ACTION _mode_manager:
IF process_mode_req_is_pending(prc)
THEN
    process_apply_mode_req_first_step(prc);
    CASE process_get_mode(prc) OF
        MODE_TO_ABSENT:
			;
        MODE_TO_INACTIVE:
			;
        MODE_TO_TEST:
			;
        MODE_TO_OPERATIONAL:
			;
    END_CASE
    process_apply_mode_req_second_step(prc);
END_IF
END_ACTION

ACTION _object_manager:
IF objects_initialization()
THEN
	sub_process_init(
		object_name					:= 'csp_case_closing_os.prc', 
		process						:= csp_case_closing.prc, 
		CONVERSION_this				:= prc);
		
	prc_path 						:= process_get_path(prc);
	
	process_message_init(
        object_name:= CONCAT(prc_path, '_Closing_paddle_Cleanout_position_aem'),
        behaviour:= MESSAGE_BEHAVIOUR_STATE,
        reset_timeout:= 0,
        disableable:= FALSE,
        individual_reset:= FALSE,
        machine_reaction:= MACHINE_REACTION_EMERGENCY_STOP, 
        typology:=  MESSAGE_TYPOLOGY_ABNORMAL,
        process:= prc,
        CONVERSION_this:= Closing_paddle_Cleanout_position_aem);
END_IF

IF objects_running()
THEN
	process_cycle(prc);
END_IF
END_ACTION

ACTION _read_process_image:
;
END_ACTION

ACTION _read_var_input:
;
END_ACTION

ACTION _set_runtime_properties:
;
END_ACTION

ACTION _write_output:
;
END_ACTION

END_PROGRAM

// ---- Application/CSP/Case/Closing/LS/csp_case_closing_ls.TcPOU
(*********************************** G.D S.p.A. - Technical Department ***********************************
============= PROGRAM INFO ============
FOLDER:             TBD
MACHINES INVOLVED:  TBD 

============= DESCRIPTION =============
csp machine declaration

============= REVISIONS ===============
Date		Version	 	Author      	Description             
----------	-------		------------  	--------------------------------------------
2019/04/05 	0000.00	 	M.Grasso		Creation of the PRG

**********************************************************************************************************)
(*$R process_ref := prc; $*)
PROGRAM csp_case_closing_ls
VAR
		
	prc:											process;
	prc_path:										STRING;
	
	phase_upper:									BOOL;
	phase_lower:									BOOL;
	phase_horizontal:								BOOL;
	
	horizontal_first:								BOOL;
	horizontal_second:								BOOL;
	
END_VAR

_read_var_input();

_object_manager();

IF NOT objects_running()
THEN
	RETURN;	
END_IF

_read_process_image();

_mode_manager();

CASE process_get_mode(prc) OF
	MODE_ABSENT,
	MODE_INACTIVE:
		RETURN;
	MODE_TEST:
		_handle_process_test();
END_CASE

_set_runtime_properties();

(********************************* BODY *********************************)

(* CLEARS PHASING SEQUENCE DUE TO AXES CAM ENGAGED *)
IF 	axis_is_cam_engaged(csp_case_closing_ls_horizontal.axis)
	OR machine_is_stop_emergency_active(csp.mch)
THEN
	phase_horizontal := FALSE;
END_IF

IF 	axis_is_cam_engaged(csp_case_closing_ls_upper.axis)
	OR machine_is_stop_emergency_active(csp.mch)
THEN
	phase_upper := FALSE;
END_IF

IF 	axis_is_cam_engaged(csp_case_closing_ls_lower.axis)
	OR machine_is_stop_emergency_active(csp.mch)
THEN
	phase_lower := FALSE;
END_IF

IF (
	axis_is_cam_engaged(csp_case_closing_ls_horizontal.axis)
	AND axis_is_cam_engaged(csp_case_closing_ls_upper.axis)
	AND axis_is_cam_engaged(csp_case_closing_ls_lower.axis)
	)
	OR machine_is_stop_emergency_active(csp.mch)
THEN
	horizontal_first := FALSE;
	horizontal_second := FALSE;
END_IF


(* HORIZONTAL NEEDS TO PHASE - CHECK IF UPPER AND LOWER MOVE FIRST OR HORIZONTAL FIRST *)
IF	NOT axis_is_cam_engaged(csp_case_closing_ls_horizontal.axis)
	AND NOT csp_case_closing_ls_horizontal.phase_done
	AND (motorization_manager_is_starting(csp_main_motorization_manager.motm) OR jog_manager_is_jog_axis_active(JOG_LIST_CSP_CASE_VIRTUAL, csp_main_jogManager.jog_manager_virtual))
THEN	
	(* CALCULATED HORIZONTAL TO MOVE IN - MOVE UPPER AND LOWER FIRST *)
	IF csp_case_closing_ls_horizontal.axis_calculated_cam_slave_position_deg >= axis_get_actual_modulo_position(csp_case_closing_ls_horizontal.axis)
	THEN
		horizontal_second := TRUE;
	(* CALCULATED HORIZONTAL TO MOVE OUT - MOVE HORIZONTAL FIRST *)
	ELSE
		horizontal_first := TRUE;
	END_IF
END_IF

(* PHASE HORIZONTAL THEN UPPER AND LOWER *)
IF 	horizontal_first
	AND (motorization_manager_is_starting(csp_main_motorization_manager.motm) OR jog_manager_is_jog_axis_active(JOG_LIST_CSP_CASE_VIRTUAL, csp_main_jogManager.jog_manager_virtual))
THEN
	phase_horizontal := TRUE;
	IF csp_case_closing_ls_horizontal.phase_done
	THEN
		phase_upper := TRUE;
		phase_lower := TRUE;
	END_IF
END_IF

(* PHASE UPPER AND LOWER THEN HORIZONTAL *)
IF horizontal_second
	AND (motorization_manager_is_starting(csp_main_motorization_manager.motm) OR jog_manager_is_jog_axis_active(JOG_LIST_CSP_CASE_VIRTUAL, csp_main_jogManager.jog_manager_virtual))
THEN
	phase_upper := TRUE;
	phase_lower := TRUE;
	IF 	csp_case_closing_ls_upper.phase_done
		AND csp_case_closing_ls_lower.phase_done
	THEN
		phase_horizontal := TRUE;
	END_IF
END_IF

(************************************************************************)

_handle_messages();

_write_output();

ACTION _handle_messages:
;
END_ACTION

ACTION _handle_process_test:
;
END_ACTION

ACTION _mode_manager:
IF process_mode_req_is_pending(prc)
THEN
    process_apply_mode_req_first_step(prc);
    CASE process_get_mode(prc) OF
        MODE_TO_ABSENT:
			;
        MODE_TO_INACTIVE:
			;
        MODE_TO_TEST:
			;
        MODE_TO_OPERATIONAL:
			;
    END_CASE
    process_apply_mode_req_second_step(prc);
END_IF
END_ACTION

ACTION _object_manager:
IF objects_initialization()
THEN
	sub_process_init(
		object_name					:= 'csp_case_closing_ls.prc', 
		process						:= csp_case_closing.prc, 
		CONVERSION_this				:= prc);
		
	prc_path 						:= process_get_path(prc);
END_IF

IF objects_running()
THEN
	process_cycle(prc);
END_IF
END_ACTION

ACTION _read_process_image:
;
END_ACTION

ACTION _read_var_input:
;
END_ACTION

ACTION _set_runtime_properties:
;
END_ACTION

ACTION _write_output:
;
END_ACTION

END_PROGRAM

// ---- Application/CSP/Case/Discharge/_Tasks/_csp_case_discharge_normal.TcPOU
(*********************************** G.D S.p.A. - Technical Department ***********************************
============= PROGRAM INFO ============
FOLDER:             TBD
MACHINES INVOLVED:  TBD 

============= DESCRIPTION =============
csp main interface program

============= REVISIONS ===============
Date		Version	 	Author      	Description             
----------	-------		------------  	--------------------------------------------
2019/09/27 	0000.00	 	M.Grasso		Creation of the PRG

**********************************************************************************************************)
PROGRAM _csp_case_discharge_normal
VAR
END_VAR

(* CASE *)
	(* DISCHARGE *)
		(* SPEEDBELT *)
		csp_case_discharge_speedBelt();
		(* REJECT *)
		csp_case_discharge_reject();

END_PROGRAM

// ---- Application/CSP/Case/Discharge/Speed Belt/csp_case_discharge_speedBelt.TcPOU
(*********************************** G.D S.p.A. - Technical Department ***********************************
============= PROGRAM INFO ============
FOLDER:             TBD
MACHINES INVOLVED:  TBD 

============= DESCRIPTION =============
csp machine declaration

============= REVISIONS ===============
Date		Version	 	Author      	Description             
----------	-------		------------  	--------------------------------------------
2019/04/05 	0000.00	 	M.Grasso		Creation of the PRG

**********************************************************************************************************)
(*$R process_ref := prc; $*)
PROGRAM csp_case_discharge_speedBelt
VAR
		
	prc:											process;
	prc_path:										STRING;
	
END_VAR

_read_var_input();

_object_manager();

IF NOT objects_running()
THEN
	RETURN;	
END_IF

_read_process_image();

_mode_manager();

_set_runtime_properties();

(********************************* BODY *********************************)
(************************************************************************)

_handle_messages();

_write_output();

ACTION _handle_messages:
;
END_ACTION

ACTION _handle_process_test:
;
END_ACTION

ACTION _mode_manager:
IF process_mode_req_is_pending(prc)
THEN
    process_apply_mode_req_first_step(prc);
    CASE process_get_mode(prc) OF
        MODE_TO_ABSENT:
			;
        MODE_TO_INACTIVE:
			;
        MODE_TO_TEST:
			;
        MODE_TO_OPERATIONAL:
			;
    END_CASE
    process_apply_mode_req_second_step(prc);
END_IF
END_ACTION

ACTION _object_manager:
IF objects_initialization()
THEN
	sub_process_init(
		object_name					:= 'csp_case_discharge_speedBelt.prc', 
		process						:= csp_case_discharge.prc, 
		CONVERSION_this				:= prc);
		
	prc_path 						:= process_get_path(prc);
END_IF

IF objects_running()
THEN
	process_cycle(prc);
END_IF
END_ACTION

ACTION _read_process_image:
;
END_ACTION

ACTION _read_var_input:
;
END_ACTION

ACTION _set_runtime_properties:
;
END_ACTION

ACTION _write_output:
;
END_ACTION

END_PROGRAM

// ---- Application/CSP/Case/Discharge/Reject/csp_case_discharge_reject.TcPOU
(*********************************** G.D S.p.A. - Technical Department ***********************************
============= PROGRAM INFO ============
FOLDER:             TBD
MACHINES INVOLVED:  TBD 

 

============= DESCRIPTION =============
csp machine declaration

 

============= REVISIONS ===============
Date        Version         Author          Description             
----------    -------        ------------      --------------------------------------------
2019/04/05     0000.00         M.Grasso        Creation of the PRG

 

**********************************************************************************************************)
(*$R process_ref := prc; $*)
PROGRAM csp_case_discharge_reject
VAR
        
    prc:                                            	process;
    prc_path:                                        	STRING;
    
    reject_ftrig:                                    	F_TRIG;
    di:                                             	Digital_input;
    reject_active:                                    	BOOL;
    reject_belt_run_delay:                             	Timer;

    status:                                         	STRING;
    start_reject:                                   	BOOL;
	trigger:                                         	BOOL;
	MODSORT_reject:                                 	BOOL;
    MODSORT_fwd:                                     	BOOL;
	reject_confirm:                                 	TON;
	start_reject_belt:                                	BOOL;
    reject_confirmed:                                 	BOOL;
    case_at_reject:                                  	INT:=28;
	open_major_LS_detected: 							BOOL := FALSE;
	open_major_OS_detected:								BOOL := FALSE;

	open_trailing_minor:								BOOL;
	Discharge_reject_count:								DINT;
	timer1:												TOF;
	timer1_value:									TIME := T#5S;
	time_complete1: 									BOOL;
	open_leading_minor: 								BOOL;
	Startup_run_ton: 									Ton;
	startup_run_condition: 								BOOL;
	modsort_belt_speed_analog_reference_ao:             analog_output;
    speed_value_nvr: 									REAL;
	stopping_run_ton: 									Ton;
	stop_run_condition: 								BOOL;
	suspend_run_ton: 									TON;
	suspend_run_condition: 								BOOL;
END_VAR
VAR CONSTANT
    MOTOR_MAX_VELOCITY_DEGPS:                        	LREAL := 9600;
    MOTOR_MIN_VELOCITY_DEGPS:                         	LREAL := 100;
    MOTOR_MAX_ACCELLERATION_DEGPS2:                    	LREAL := 4800;
    MOTOR_MAX_DECELLERATION_DEGPS2:                    	LREAL := 4800;
    MOTOR_MAX_JERK_DEGPS3:                            	LREAL := 100000000; 
    MOTOR_MAX_FOLLOWING_ERROR_DEG:                    	LREAL := 2;
END_VAR

_read_var_input();

 

_object_manager();

 

IF NOT objects_running()
THEN
    RETURN;    
END_IF

 

_read_process_image();

 

_mode_manager();

 

_set_runtime_properties();

 

(********************************* BODY *********************************)
(* Handles stops for reject belt and Modsort Motors to turnoff when machine is not in execute *)
IF  (
	axis_is_moving(csp_main_motorization_virtualManager.axis) 
	OR 
	NOT stop_run_condition
	)
	AND NOT csp.o_machine_is_emergency_stopped
THEN 
 	speed_value_nvr := csp_main_motorization_manager.motm.actual_velocity * 200;
ELSE
	speed_value_nvr := 0;
END_IF

analog_output_electrical_write(
    electrical_value := speed_value_nvr,
    conversion_THIS := modsort_belt_speed_analog_reference_ao);
 
IF 	reject_confirmed
THEN
    modsort_reject := FALSE;
    digital_output_reset(conversion_this:= csp_case_discharge_reject_modsort.MODSORT_REJECT_RUN_do); //stops modosort when machine is stopped
END_IF

(*Latches in open flap detected when in window and open flap PE is blocked *)
IF 	((csp_case_virtualMaster.axis.actual_position > csp_case_openFlap_sensors.OpenMajorFlapChkBeginPhase)
	AND
	(csp_case_virtualMaster.axis.actual_position < csp_case_openFlap_sensors.OpenMajorFlapChkEndPhase))
THEN
	IF	NOT digital_input_is_active(csp_case_openFlap_sensors.open_flap_ls_di)
	THEN
		open_major_LS_detected :=TRUE;
	END_IF
	
	IF	NOT digital_input_is_active(csp_case_openFlap_sensors.open_flap_os_di)
	THEN
		open_major_OS_detected :=TRUE;
	END_IF
 END_IF
 
 
(* Resets open flap detected latch *)
IF 	open_major_LS_detected
 	AND axis_get_actual_modulo_position(csp_case_transport_virtualMaster.axis) > 350 //resets open major detected before next case
THEN
	open_major_LS_detected := FALSE;
END_IF

(* Resets open flap detected latch *)
IF 	open_major_OS_detected
 	AND axis_get_actual_modulo_position(csp_case_transport_virtualMaster.axis) > 350 //resets open major detected before next case
THEN
	open_major_OS_detected := FALSE;
END_IF

(* LATCHES BIT FOR OPEN TRAILING MINOR *)
IF 	csp_case_transport_virtualMaster.axis.actual_position > csp_case_openFlap_sensors.open_trailing_minor_begin_phase
	AND csp_case_transport_virtualMaster.axis.actual_position < csp_case_openFlap_sensors.open_trailing_minor_end_phase
THEN
	IF digital_input_is_active(csp_case_openFlap_sensors.open_trailing_minor_di)
	THEN
		open_trailing_minor := TRUE;
	END_IF
END_IF

(* Resets open trailing minor detected latch *)
IF 	open_trailing_minor
	AND axis_get_actual_modulo_position(csp_case_transport_virtualMaster.axis) > 350 //resets open major detected before next case
THEN
 	open_trailing_minor := FALSE;
END_IF

(* LATCHES BIT FOR OPEN LEADING MINOR *)
IF 	csp_case_transport_virtualMaster.axis.actual_position > csp_case_openFlap_sensors.open_leading_minor_begin_phase
	AND csp_case_transport_virtualMaster.axis.actual_position < csp_case_openFlap_sensors.open_leading_minor_end_phase
THEN
	IF digital_input_is_active(csp_case_openFlap_sensors.open_trailing_minor_di)
	THEN
		open_leading_minor := TRUE;
	END_IF
END_IF

(* Resets open OPEN LEADING MINOR detected latch *)
IF 	open_leading_minor
	AND axis_get_actual_modulo_position(csp_case_transport_virtualMaster.axis) > 350 //resets open major detected before next case
THEN
 	open_leading_minor := FALSE;
END_IF

(* Sets shift register if detected *)
IF open_trailing_minor
THEN
	shift_register_step_set_reject_reason(
		reject_reason_to_set := TRAILING_MINOR_FLAP_OPEN,
		step_id := 28,
		CONVERSION_this := csp_case_main_statistics.sr);
END_IF

(* Sets shift register if detected *)
IF 	open_leading_minor
THEN
	shift_register_step_set_reject_reason(
		reject_reason_to_set := LEADING_MINOR_FLAP_OPEN,
		step_id := 28,
		CONVERSION_this := csp_case_main_statistics.sr);
END_IF

(* Sets shift register if detected *)
IF 	open_major_LS_detected
THEN
	shift_register_step_set_reject_reason(
		reject_reason_to_set := OPEN_FLAP_LOADER_SIDE,
		step_id := 28,
		CONVERSION_this := csp_case_main_statistics.sr);
END_IF

(* Sets shift register if detected *)
IF 	open_major_OS_detected
THEN	
	shift_register_step_set_reject_reason(
		reject_reason_to_set := OPEN_FLAP_OPERATOR_SIDE,
		step_id := 28,
		CONVERSION_this := csp_case_main_statistics.sr);
END_IF

(* Shift Register detects if there is a reject *)
IF shift_register_step_has_any_reject_reason(
	step_id:= case_at_reject, 
	CONVERSION_this:= csp_case_main_statistics.sr)
THEN
	reject_active := TRUE;
ELSE
	reject_active:= FALSE;
END_IF
             
digital_input_read(trigger, csp_case_discharge_reject_sensors.reject_trigger_di); // sets 'trigger' as bool for digital input OF PhotoEye

reject_ftrig(CLK := trigger); // falling edge of trigger //starts reject on trigger if reject_active (ON)

reject_confirm(IN:=start_reject , PT:=T#2S , Q=> reject_confirmed , ET=> );// how long to run reject operation or setup with Photoeye for confirmation

IF reject_active AND reject_ftrig.Q    //start sequence when PE triggered
THEN
	start_reject := TRUE;
END_IF
    
(* Resets start_reject to end the reject sequence *)    
IF reject_confirmed 
THEN     (*resets bit when reject confirmed (2 Second Timer); works for max speed at 27.5 cpm with cycle being 2.18 seconds *)
    start_reject := FALSE;    
END_IF            

(********************************* MODSORT LOGIC *********************************)
stopping_run_ton(IN:= NOT axis_is_moving(csp_main_motorization_virtualManager.axis) , PT:=T#10S , Q=> stop_run_condition , ET=> );
suspend_run_ton(
				IN:= motorization_manager_is_held(csp_main_motorization_manager.motm) OR motorization_manager_is_suspended(csp_main_motorization_manager.motm),
				PT:=T#20S,
				Q=> suspend_run_condition,
				ET=> );
 
IF 	(
		(
			axis_is_moving(csp_main_motorization_virtualManager.axis) 
			OR
			NOT stop_run_condition //becomes true after moto VM stopped for 2 seconds
		)
		AND NOT suspend_run_condition //becomes true after 5 seconds of being in suspend or held state
	)
	AND NOT csp.o_machine_is_emergency_stopped
THEN
	IF digital_output_is_active(conversion_this:= csp_case_discharge_reject_modsort.MODSORT_REJECT_RUN_do)
	THEN
		digital_output_reset(conversion_this:= csp_case_discharge_reject_modsort.MODSORT_FWD_RUN_do);
		modsort_fwd := FALSE; //testing
	ELSE
		modsort_fwd := TRUE; //testing
		digital_output_set(conversion_this:= csp_case_discharge_reject_modsort.MODSORT_FWD_RUN_do);
	END_IF    
ELSE
	modsort_fwd := FALSE; //testing
	digital_output_reset(conversion_this:= csp_case_discharge_reject_modsort.MODSORT_FWD_RUN_do);
END_IF

(* If reject sequence activated, and machine running, then run modsort reject motor until confirmed with (2 second) timer.*)    
IF 	reject_active 
	AND start_reject 
	AND NOT reject_confirmed    //reject once started until reject_confirm TRUE
THEN
	modsort_reject := TRUE;
	digital_output_set(conversion_this:= csp_case_discharge_reject_modsort.MODSORT_REJECT_RUN_do);
END_IF    
    
start_reject_belt := reject_active//start_reject                             //conditions for starting reject belt
                    OR digital_output_is_active(conversion_this:= csp_case_discharge_reject_modsort.MODSORT_REJECT_RUN_do);          
        

(********************************* Belt Run duration *********************************)
							
timer1.IN := trigger;
time_complete1 := NOT timer1.Q;
timer1(PT := timer1_value);

(********************************* REJECT BELT LOGIC *********************************)
Startup_run_ton(IN:=axis_is_moving(csp_main_motorization_virtualManager.axis) , PT:=T#5S , Q=> startup_run_condition , ET=> );

IF 	(
		start_reject_belt 
		AND NOT time_complete1
	)
	OR
	(
		axis_is_moving(csp_main_motorization_virtualManager.axis)
		AND NOT startup_run_condition
	)
THEN
	axis_set_override(                        //overides axis velocity to the set JOG speed, JOG set at 10 in csp_case_discharge_belts_conveyor (TEST SPEED - Austin)
		speed_override_percent     := 30,
		CONVERSION_this         := csp_case_discharge_reject_belt.axis);//csp_case_discharge_belts_conveyor.axis
	status := 'Belt moving';
ELSE
	axis_set_override(          
		speed_override_percent     := 0,
		CONVERSION_this         := csp_case_discharge_reject_belt.axis);
	status := 'Stopped';
END_IF


(************************************************************************)

Discharge_Reject_Count :=
(
csp_case_main_statistics.logsect.hmi_shift_independent_sampled_counters.reject_reasons_counters[16]
+
csp_case_main_statistics.logsect.hmi_shift_independent_sampled_counters.reject_reasons_counters[17]
+
csp_case_main_statistics.logsect.hmi_shift_independent_sampled_counters.reject_reasons_counters[18]
+
csp_case_main_statistics.logsect.hmi_shift_independent_sampled_counters.reject_reasons_counters[19]
+
csp_case_main_statistics.logsect.hmi_shift_independent_sampled_counters.reject_reasons_counters[20]
+
csp_case_main_statistics.logsect.hmi_shift_independent_sampled_counters.reject_reasons_counters[21]
+
csp_case_main_statistics.logsect.hmi_shift_independent_sampled_counters.reject_reasons_counters[22]
+
csp_case_main_statistics.logsect.hmi_shift_independent_sampled_counters.reject_reasons_counters[23]
+
csp_case_main_statistics.logsect.hmi_shift_independent_sampled_counters.reject_reasons_counters[24]
);
(************************************************************************)


 

_handle_messages();

 

_write_output();

ACTION _handle_messages:
;
END_ACTION

ACTION _handle_process_test:
;
END_ACTION

ACTION _mode_manager:
IF process_mode_req_is_pending(prc)
THEN
    process_apply_mode_req_first_step(prc);
    CASE process_get_mode(prc) OF
        MODE_TO_ABSENT:
			;
        MODE_TO_INACTIVE:
			;
        MODE_TO_TEST:
			;
        MODE_TO_OPERATIONAL:
			;
    END_CASE
    process_apply_mode_req_second_step(prc);
END_IF
END_ACTION

ACTION _object_manager:
IF objects_initialization()
THEN
	sub_process_init(
		object_name					:= 'csp_case_discharge_reject.prc', 
		process						:= csp_case_discharge.prc, 
		CONVERSION_this				:= prc);
		
	prc_path 						:= process_get_path(prc);
	
	timer_init(
    	object_name:= 'csp_case_discharge_reject.reject_belt_run_delay',
    	process:= prc,
    	conversion_THIS:= reject_belt_run_delay);

 analog_output_init(
            object_name            	:= '_modsort_belt_speed_analog_reference_ao',
            field_min            	:= 0,                                (* Campo lettura modulo Beckhoff, unità - min value *)
            field_max             	:= MAX_INT_VALUE,                    (* Campo lettura modulo Beckhoff, unità - max value *)
            field_ele_xa        	:= 0,
            field_ele_ya        	:= 0,
            field_ele_xb        	:= MAX_INT_VALUE,
            field_ele_yb        	:= 10000,
            electrical_min        	:= 0,                                (* Saturazione - valore minimo in uscita, mV *)
            electrical_max        	:= 10000,                            (* Saturazione - valore massimo in uscita, mV *)
            ele_phy_xa           	:= 0,        (* mV *)
            ele_phy_ya            	:= 0,        (* PPM *)
            ele_phy_xb            	:= 10000,    (* mV *)
            ele_phy_yb            	:= 10000,    (* PPM *)
            physical_min        	:= 0,        (* rpm *)
            physical_max         	:= 5000,    (* rpm *)
            process                	:= prc,
            conversion_THIS         := modsort_belt_speed_analog_reference_ao
            ); 
END_IF

IF objects_running()
THEN
	process_cycle(prc);
    analog_output_cycle(conversion_THIS := modsort_belt_speed_analog_reference_ao);
END_IF
END_ACTION

ACTION _read_process_image:
;
END_ACTION

ACTION _read_var_input:
;
END_ACTION

ACTION _set_runtime_properties:
;
END_ACTION

ACTION _write_output:
;
END_ACTION

END_PROGRAM

// ---- Application/CSP/Case/Open Flap/Sensors/csp_case_openFlap_sensors.TcPOU
(*********************************** G.D S.p.A. - Technical Department ***********************************
============= PROGRAM INFO ============
FOLDER:             TBD
MACHINES INVOLVED:  TBD 

============= DESCRIPTION =============
csp machine declaration

============= REVISIONS ===============
Date		Version	 	Author      	Description             
----------	-------		------------  	--------------------------------------------
2019/04/05 	0000.00	 	M.Grasso		Creation of the PRG

**********************************************************************************************************)
(*$R process_ref := prc; $*)
PROGRAM csp_case_openFlap_sensors
VAR
	
	prc:											process;
	prc_path:										STRING;
	
	open_flap_ls_di:								digital_input;
	open_flap_os_di:								digital_input;
		
	open_major_flap_os_di_dchk: 					check_section;
	open_major_flap_ls_di_dchk: 					check_section;
	
	
	open_trailing_minor_di:							digital_input;
	open_trailing_minor_chksect:					check_section;
	open_trailing_minor_begin_phase: 				LREAL := 170; (*$P $*)
	open_trailing_minor_end_phase:					LREAL := 188; (*$P $*)
	
	open_leading_minor_chksect:						check_section;
	open_leading_minor_begin_phase: 				LREAL := 90; (*$P $*)
	open_leading_minor_end_phase:					LREAL := 110; (*$P $*)
	
	quality_reject_dchk: 							check_section;
	quality_reject_bool: 							boolean;
	quality_reject_req:								BOOL:= FALSE; (*$P $*)
	quality_reject_aem:								message;
	
	incomplete_glue_reject_dchk: 					check_section;
	incomplete_glue_reject_bool: 					boolean;
	incomplete_glue_reject_aem:						message;
	incomplete_glue_begin_phase: 					LREAL := 10; (*$P $*)
	incomplete_glue_end_phase:						LREAL := 300; (*$P $*)
	
	
	OpenMajorFlapChkBeginPhase: 					LREAL :=100;(*$P $*)
	OpenMajorFlapChkEndPhase:						LREAL :=350;(*$P $*)
	majorFlap_os_inchoerence_chksect: 				check_section;
	majorFlap_ls_inchoerence_chksect: 				check_section;
	
	incomplete_glue_reject: 						BOOL;
	check_step_nvr: 								DINT := 26;
	
	detect_next_case_edges: 						BOOL;(*$P desc:= DETECT LEADING AND TRAILING PHASE OF NEXT CASE; $*)
	eye_test_temp: 									BOOL;
	detected_case_leading_edge: 					LREAL;(*$P desc:= DETECTED LEADING PHASE OF CASE; $*)
	detected_case_trailing_edge: 					LREAL;(*$P desc:= DETECTED TRAILING PHASE OF CASE; $*)
END_VAR

_read_var_input();

_object_manager();

IF NOT objects_running()
THEN
	RETURN;	
END_IF

_read_process_image();

_mode_manager();

_set_runtime_properties();

(********************************* BODY *********************************)
check_section_set_check_window_phases_value(
    begin_phase         :=  OpenMajorFlapChkBeginPhase,
    end_phase           :=  OpenMajorFlapChkEndPhase,
    conversion_THIS     :=  open_major_flap_os_di_dchk);

check_section_set_check_window_phases_value(
    begin_phase         :=  OpenMajorFlapChkBeginPhase,
    end_phase           :=  OpenMajorFlapChkEndPhase,
    conversion_THIS     :=  open_major_flap_ls_di_dchk);	
	
	
check_section_set_check_window_phases_value(
    begin_phase         :=  open_trailing_minor_begin_phase,
    end_phase           :=  open_trailing_minor_end_phase,
    conversion_THIS     :=  open_trailing_minor_chksect);	

check_section_set_check_window_phases_value(
    begin_phase         :=  open_leading_minor_begin_phase,
    end_phase           :=  open_leading_minor_end_phase,
    conversion_THIS     :=  open_leading_minor_chksect);		
	
IF quality_reject_req //quality check pb on hmi to reject a case for inspection. Uses checksection to look for pb and then trigger the reject
THEN
	boolean_set(quality_reject_bool);
ELSE
	boolean_reset(quality_reject_bool);
END_IF

//checks for motion and Emergency stop to reject 
check_section_set_check_window_phases_value(
	begin_phase := incomplete_glue_begin_phase,
	end_phase := incomplete_glue_end_phase,
	CONVERSION_this := incomplete_glue_reject_dchk); 

IF check_section_get_step(incomplete_glue_reject_dchk) <> check_step_nvr
THEN
	check_section_set_step(check_step_nvr, incomplete_glue_reject_dchk);
END_IF

IF 	axis_get_actual_modulo_position(csp_case_transport_virtualMaster.axis) > incomplete_glue_begin_phase  
	AND axis_get_actual_modulo_position(csp_case_transport_virtualMaster.axis) < incomplete_glue_end_phase  
	AND machine_is_stop_emergency_active(csp.mch)
THEN
	boolean_set(incomplete_glue_reject_bool);
	incomplete_glue_reject := TRUE ;
END_IF

IF axis_get_actual_modulo_position(csp_case_transport_virtualMaster.axis) > 359
THEN
	boolean_reset(incomplete_glue_reject_bool);
	incomplete_glue_reject := FALSE ;
END_IF

IF csp_case_main_services.dry_cycle_mode
	OR csp_main_motorization.empty_command
THEN
	check_section_disable(majorFlap_os_inchoerence_chksect);
	check_section_disable(majorFlap_ls_inchoerence_chksect);
	check_section_disable(open_major_flap_os_di_dchk);
	check_section_disable(open_major_flap_ls_di_dchk);
	check_section_disable(open_trailing_minor_chksect);
	check_section_disable(open_leading_minor_chksect);
ELSE
	check_section_enable(majorFlap_os_inchoerence_chksect);
	check_section_enable(majorFlap_ls_inchoerence_chksect);
	check_section_enable(open_major_flap_os_di_dchk);
	check_section_enable(open_major_flap_ls_di_dchk);
	check_section_enable(open_trailing_minor_chksect);
	check_section_enable(open_leading_minor_chksect);
END_IF		


IF quality_reject_req
THEN
	process_message_set(1, 1, 1, quality_reject_aem);
ELSE
	process_message_reset(quality_reject_aem);
END_IF

(* Turn on eye_test to capture the leading and trailing edge of the box as it passes open-flap eye. Use these values to then set appropriate phase window values for open flap detection. *)
IF 	detect_next_case_edges
	AND NOT eye_test_temp
	AND digital_input_is_active(open_trailing_minor_di)
then
	detected_case_leading_edge := csp_case_transport_virtualMaster.axis.actual_position;
	eye_test_temp := TRUE;
	detect_next_case_edges := FALSE;
end_if

IF 	eye_test_temp
	AND NOT digital_input_is_active(open_trailing_minor_di)
then
	detected_case_trailing_edge := csp_case_transport_virtualMaster.axis.actual_position;
	eye_test_temp := FALSE;
end_if
(************************************************************************)

_handle_messages();

_write_output();

ACTION _handle_messages:
;
END_ACTION

ACTION _handle_process_test:
;
END_ACTION

ACTION _mode_manager:
IF process_mode_req_is_pending(prc)
THEN
    process_apply_mode_req_first_step(prc);
    CASE process_get_mode(prc) OF
        MODE_TO_ABSENT:
			;
        MODE_TO_INACTIVE:
			;
        MODE_TO_TEST:
			;
        MODE_TO_OPERATIONAL:
			;
    END_CASE
    process_apply_mode_req_second_step(prc);
END_IF
END_ACTION

ACTION _object_manager:
IF objects_initialization()
THEN
    sub_process_init(
        object_name                    := 'csp_case_openFlap_sensors.prc',
        process                        := csp_case_openFlap.prc,
        CONVERSION_this                := prc);
       
    prc_path                         := process_get_path(prc);
   
    (* INPUTS *)
    digital_input_init(
        object_name                    := CONCAT(prc_path, '_open_flap_ls_di'),
        polarity_direct                := TRUE,
        process                        := prc,
        CONVERSION_this                := open_flap_ls_di);
       
    digital_input_init(
        object_name                    := CONCAT(prc_path, '_open_flap_os_di'),
        polarity_direct                := TRUE,
        process                        := prc,
        CONVERSION_this                := open_flap_os_di);
		
	digital_input_init(
        object_name                    := CONCAT(prc_path, '_open_trailing_minor_di'),
        polarity_direct                := TRUE,
        process                        := prc,
        CONVERSION_this                := open_trailing_minor_di);
  
		
	 boolean_init(
		object_name 				   := CONCAT(prc_path, '_quality_reject_bool'),
		process 			   		   := prc,
		CONVERSION_this				   := quality_reject_bool);
	
	 boolean_init(
		object_name 				   := CONCAT(prc_path, '_incomplete_glue_reject_bool'),
		process 					   := prc,
		CONVERSION_this				   := incomplete_glue_reject_bool);

		
		
(*OPEN FLAP OPERATOR SIDE SENSOR LOGIC*)  
	check_section_window_mode_init(
		object_name:= CONCAT(prc_path, '_open_major_flap_os_di_dchk'),
		check_enable:= TRUE, 
		event_to_check:= CHECK_SECTION_EVENT_INPUT_OFF, 
		execution_mode:= CHECK_SECTION_EXECUTION_WHEN_EVENT_OCCURRED, 
		diagnostic_enable:= FALSE, 
		status_bits_to_be_true:= ITEM_CASE_FEED, 
		status_bits_to_be_false:= 0, 
		_step_status_conditioning_execution:= FALSE, 
		status_bits_to_set:= OPEN_FLAP_OPERATOR_SIDE, 
		status_bits_to_reset:= 0, 
		reject_bit_to_set:= OPEN_FLAP_OPERATOR_SIDE, 
		_step:= 28, 
		first_step_to_write_offset:= 0, 
		number_of_steps_to_write:= 1, 
		begin_phase:= OpenMajorFlapChkBeginPhase, 
		end_phase:= OpenMajorFlapChkEndPhase, 
		max_consecutive_failed_checks:= 3, 
		max_failed_checks_percentage:= 100, 
		products_for_failed_checks_percentage:= 10, 
		shift_register:= csp_case_main_statistics.sr , 
		process:= prc, 
		CONVERSION_this:= open_major_flap_os_di_dchk );

	check_section_add_di_input(
		di_input := open_flap_os_di,
		CONVERSION_this:= open_major_flap_os_di_dchk);
	
	message_configure(
        individual_reset                    := FALSE,
        machine_reaction                    := MACHINE_REACTION_STOP_IN_PHASE_ONE,
        typology                            := MESSAGE_TYPOLOGY_ABNORMAL,
        CONVERSION_this                     := open_major_flap_os_di_dchk.too_many_failed_checks_aem.message );	
	
	
 (*OPEN FLAP LOADER SIDE SENSOR LOGIC*)  
	check_section_window_mode_init(
		object_name:= CONCAT(prc_path, '_open_major_flap_ls_di_dchk'),
		check_enable:= TRUE, 
		event_to_check:= CHECK_SECTION_EVENT_INPUT_OFF, 
		execution_mode:= CHECK_SECTION_EXECUTION_WHEN_EVENT_OCCURRED, 
		diagnostic_enable:= FALSE, 
		status_bits_to_be_true:= ITEM_CASE_FEED, 
		status_bits_to_be_false:= 0, 
		_step_status_conditioning_execution:= FALSE, 
		status_bits_to_set:= OPEN_FLAP_LOADER_SIDE, 
		status_bits_to_reset:= 0, 
		reject_bit_to_set:= OPEN_FLAP_LOADER_SIDE, 
		_step:= 28, 
		first_step_to_write_offset:= 0, 
		number_of_steps_to_write:= 1, 
		begin_phase:= OpenMajorFlapChkBeginPhase, 
		end_phase:= OpenMajorFlapChkEndPhase, 
		max_consecutive_failed_checks:= 3, 
		max_failed_checks_percentage:= 100, 
		products_for_failed_checks_percentage:= 10, 
		shift_register:= csp_case_main_statistics.sr , 
		process:= prc, 
		CONVERSION_this:= open_major_flap_ls_di_dchk );

	check_section_add_di_input(
		di_input := open_flap_ls_di,
		CONVERSION_this:= open_major_flap_ls_di_dchk);	
    
	message_configure(
        individual_reset                    := FALSE,
        machine_reaction                    := MACHINE_REACTION_STOP_IN_PHASE_ONE,
        typology                            := MESSAGE_TYPOLOGY_ABNORMAL,
        CONVERSION_this                     := open_major_flap_ls_di_dchk.too_many_failed_checks_aem.message );	
	
    
	(*Quality Reject SENSOR LOGIC*)  //added for quality reject push button on hmi
	check_section_window_mode_init(
		object_name:= CONCAT(prc_path, '_quality_reject_dchk'),
		check_enable:= TRUE, 
		event_to_check:= CHECK_SECTION_EVENT_INPUT_ON, 
		execution_mode:= CHECK_SECTION_EXECUTION_WHEN_EVENT_OCCURRED, 
		diagnostic_enable:= FALSE, 
		status_bits_to_be_true:= ITEM_CASE_FEED, 
		status_bits_to_be_false:= 0, 
		_step_status_conditioning_execution:= FALSE, 
		status_bits_to_set:= 0, 
		status_bits_to_reset:= 0, 
		reject_bit_to_set:= QUALITY_REJECT, 
		_step:= 28, 
		first_step_to_write_offset:= 0, 
		number_of_steps_to_write:= 1, 
		begin_phase:= 10, 
		end_phase:= 340, 
		max_consecutive_failed_checks:= 3, 
		max_failed_checks_percentage:= 100, 
		products_for_failed_checks_percentage:= 10, 
		shift_register:= csp_case_main_statistics.sr , 
		process:= prc, 
		CONVERSION_this:= quality_reject_dchk );

	check_section_add_boolean_input(
		boolean_input:= quality_reject_bool,
		CONVERSION_this:= quality_reject_dchk);	
		
	message_configure(
        individual_reset                    := FALSE,
        machine_reaction                    := MACHINE_REACTION_STOP_IN_PHASE_ONE,
        typology                            := MESSAGE_TYPOLOGY_ABNORMAL,
        CONVERSION_this                     := quality_reject_dchk.too_many_failed_checks_aem.message );		
		
	
check_section_window_mode_init(
		object_name:= CONCAT(prc_path, '_majorFlap_os_inchoerence_chksect'),
		check_enable:= TRUE, 
		event_to_check:= CHECK_SECTION_EVENT_INPUT_ALWAYS_ON, 
		execution_mode:= CHECK_SECTION_EXECUTION_WHEN_EVENT_NOT_OCCURRED, 
		diagnostic_enable:= FALSE, 
		status_bits_to_be_true:= ITEM_CASE_FEED, 
		status_bits_to_be_false:= 0, 
		_step_status_conditioning_execution:= FALSE, 
		status_bits_to_set:= 0, 
		status_bits_to_reset:= 0, 
		reject_bit_to_set:= OPEN_FLAP_OPERATOR_SIDE_INCHOERENCE, 
		_step:= 28, 
		first_step_to_write_offset:= 0, 
		number_of_steps_to_write:= 1, 
		begin_phase:= csp_case_flapControl.Flap_check_begin_phase, 
		end_phase:= csp_case_flapControl.Flap_check_end_phase, 
		max_consecutive_failed_checks:= 3, 
		max_failed_checks_percentage:= 100, 
		products_for_failed_checks_percentage:= 99, 
		shift_register:= csp_case_main_statistics.sr , 
		process:= prc, 
		CONVERSION_this:= majorFlap_os_inchoerence_chksect );

	check_section_add_di_input(
		di_input := open_flap_os_di,
		CONVERSION_this:= majorFlap_os_inchoerence_chksect);

	message_configure(
        individual_reset                    := FALSE,
        machine_reaction                    := MACHINE_REACTION_STOP_IN_PHASE_ONE,
        typology                            := MESSAGE_TYPOLOGY_ABNORMAL,
        CONVERSION_this                     := majorFlap_os_inchoerence_chksect.too_many_failed_checks_aem.message );	
		
    check_section_window_mode_init(
		object_name:= CONCAT(prc_path, '_majorFlap_ls_inchoerence_chksect'),
		check_enable:= TRUE, 
		event_to_check:= CHECK_SECTION_EVENT_INPUT_ALWAYS_ON, 
		execution_mode:= CHECK_SECTION_EXECUTION_WHEN_EVENT_NOT_OCCURRED, 
		diagnostic_enable:= FALSE, 
		status_bits_to_be_true:= ITEM_CASE_FEED, 
		status_bits_to_be_false:= 0, 
		_step_status_conditioning_execution:= FALSE, 
		status_bits_to_set:= 0, 
		status_bits_to_reset:= 0, 
		reject_bit_to_set:= OPEN_FLAP_LOADER_SIDE_INCHOERENCE, 
		_step:= 28, 
		first_step_to_write_offset:= 0, 
		number_of_steps_to_write:= 1, 
		begin_phase:= csp_case_flapControl.Flap_check_begin_phase, 
		end_phase:= csp_case_flapControl.Flap_check_end_phase, 
		max_consecutive_failed_checks:= 3, 
		max_failed_checks_percentage:= 100, 
		products_for_failed_checks_percentage:= 99, 
		shift_register:= csp_case_main_statistics.sr , 
		process:= prc, 
		CONVERSION_this:= majorFlap_ls_inchoerence_chksect );

	check_section_add_di_input(
		di_input := open_flap_ls_di,
		CONVERSION_this:= majorFlap_ls_inchoerence_chksect);
		
	message_configure(
        individual_reset                    := FALSE,
        machine_reaction                    := MACHINE_REACTION_STOP_IN_PHASE_ONE,
        typology                            := MESSAGE_TYPOLOGY_ABNORMAL,
        CONVERSION_this                     := majorFlap_ls_inchoerence_chksect.too_many_failed_checks_aem.message );		
		
	
	(* OPEN TRAILING MINOR LOGIC *)
	check_section_window_mode_init(
		object_name:= CONCAT(prc_path, '_open_trailing_minor_chksect'),
		check_enable:= TRUE, 
		event_to_check:= CHECK_SECTION_EVENT_INPUT_ALWAYS_OFF, 
		execution_mode:= CHECK_SECTION_EXECUTION_WHEN_EVENT_NOT_OCCURRED, 
		diagnostic_enable:= FALSE, 
		status_bits_to_be_true:= ITEM_CASE_FEED, 
		status_bits_to_be_false:= 0, 
		_step_status_conditioning_execution:= FALSE, 
		status_bits_to_set:= 0, 
		status_bits_to_reset:= 0, 
		reject_bit_to_set:= TRAILING_MINOR_FLAP_OPEN, 
		_step:= 28, 
		first_step_to_write_offset:= 0, 
		number_of_steps_to_write:= 1, 
		begin_phase:= open_trailing_minor_begin_phase, 
		end_phase:= open_trailing_minor_end_phase, 
		max_consecutive_failed_checks:= 3, 
		max_failed_checks_percentage:= 100, 
		products_for_failed_checks_percentage:= 99, 
		shift_register:= csp_case_main_statistics.sr , 
		process:= prc, 
		CONVERSION_this:= open_trailing_minor_chksect);

	check_section_add_di_input(
		di_input := open_trailing_minor_di,
		CONVERSION_this:= open_trailing_minor_chksect);
	
	message_configure(
        individual_reset                    := FALSE,
        machine_reaction                    := MACHINE_REACTION_STOP_IN_PHASE_ONE,
        typology                            := MESSAGE_TYPOLOGY_ABNORMAL,
        CONVERSION_this                     := open_trailing_minor_chksect.too_many_failed_checks_aem.message );	
	
	(* OPEN LEADING MINOR LOGIC *)
	check_section_window_mode_init(
		object_name:= CONCAT(prc_path, '_open_leading_minor_chksect'),
		check_enable:= TRUE, 
		event_to_check:= CHECK_SECTION_EVENT_INPUT_ALWAYS_OFF, 
		execution_mode:= CHECK_SECTION_EXECUTION_WHEN_EVENT_NOT_OCCURRED, 
		diagnostic_enable:= FALSE, 
		status_bits_to_be_true:= ITEM_CASE_FEED, 
		status_bits_to_be_false:= 0, 
		_step_status_conditioning_execution:= FALSE, 
		status_bits_to_set:= 0, 
		status_bits_to_reset:= 0, 
		reject_bit_to_set:= LEADING_MINOR_FLAP_OPEN, 
		_step:= 28, 
		first_step_to_write_offset:= 0, 
		number_of_steps_to_write:= 1, 
		begin_phase:= open_leading_minor_begin_phase, 
		end_phase:= open_leading_minor_end_phase, 
		max_consecutive_failed_checks:= 3, 
		max_failed_checks_percentage:= 100, 
		products_for_failed_checks_percentage:= 99, 
		shift_register:= csp_case_main_statistics.sr , 
		process:= prc, 
		CONVERSION_this:= open_leading_minor_chksect);

	check_section_add_di_input(
		di_input := open_trailing_minor_di,
		CONVERSION_this:= open_leading_minor_chksect); 
    
	message_configure(
        individual_reset                    := FALSE,
        machine_reaction                    := MACHINE_REACTION_STOP_IN_PHASE_ONE,
        typology                            := MESSAGE_TYPOLOGY_ABNORMAL,
        CONVERSION_this                     := open_leading_minor_chksect.too_many_failed_checks_aem.message );	
		
    
		(*Emergency Stop Reject Logic*)  //added for glue
	check_section_window_mode_init(
		object_name:= CONCAT(prc_path, '_incomplete_glue_reject_dchk'),
		check_enable:= TRUE, 
		event_to_check:= CHECK_SECTION_EVENT_INPUT_ON, 
		execution_mode:= CHECK_SECTION_EXECUTION_WHEN_EVENT_OCCURRED, 
		diagnostic_enable:= FALSE, 
		status_bits_to_be_true:= ITEM_CASE_FEED, 
		status_bits_to_be_false:= 0, 
		_step_status_conditioning_execution:= FALSE, 
		status_bits_to_set:= 0, 
		status_bits_to_reset:= 0, 
		reject_bit_to_set:= INCOMPLETE_GLUE, 
		_step:= 28, 
		first_step_to_write_offset:= 0, 
		number_of_steps_to_write:= 1, 
		begin_phase:= 10, 
		end_phase:= 340, 
		max_consecutive_failed_checks:= 3, 
		max_failed_checks_percentage:= 100, 
		products_for_failed_checks_percentage:= 10, 
		shift_register:= csp_case_main_statistics.sr , 
		process:= prc, 
		CONVERSION_this:= incomplete_glue_reject_dchk );

	check_section_add_boolean_input(
		boolean_input:= incomplete_glue_reject_bool,
		CONVERSION_this:= incomplete_glue_reject_dchk);			
		
	message_configure(
        individual_reset                    := FALSE,
        machine_reaction                    := MACHINE_REACTION_STOP_IN_PHASE_ONE,
        typology                            := MESSAGE_TYPOLOGY_ABNORMAL,
        CONVERSION_this                     := incomplete_glue_reject_dchk.too_many_failed_checks_aem.message );			
		
	process_message_init(
		object_name					:=	CONCAT(prc_path, '_quality_reject_aem'), 
		behaviour					:=	MESSAGE_BEHAVIOUR_STATE,
		reset_timeout				:=	0,
		disableable					:=	TRUE,
		individual_reset			:=	FALSE,
		machine_reaction			:=	MACHINE_REACTION_NO_STOP,
		typology					:=	MESSAGE_TYPOLOGY_GENERIC_1,
		process						:=	prc,
		CONVERSION_this				:=	quality_reject_aem);
   
	process_message_init(
		object_name					:=	CONCAT(prc_path, '_incomplete_glue_reject_aem'), 
		behaviour					:=	MESSAGE_BEHAVIOUR_STATE,
		reset_timeout				:=	0,
		disableable					:=	TRUE,
		individual_reset			:=	FALSE,
		machine_reaction			:=	MACHINE_REACTION_NO_STOP,
		typology					:=	MESSAGE_TYPOLOGY_GENERIC_1,
		process						:=	prc,
		CONVERSION_this				:=	incomplete_glue_reject_aem);    
END_IF


IF objects_running()
THEN
    process_cycle(prc);
    
END_IF
END_ACTION

ACTION _read_process_image:
;
END_ACTION

ACTION _read_var_input:
;
END_ACTION

ACTION _set_runtime_properties:

END_ACTION

ACTION _write_output:
;
END_ACTION

END_PROGRAM

// ---- Application/CSP/Case/Feed/_Tasks/_csp_case_feed_normal.TcPOU
(*********************************** G.D S.p.A. - Technical Department ***********************************
============= PROGRAM INFO ============
FOLDER:             TBD
MACHINES INVOLVED:  TBD 

============= DESCRIPTION =============
csp main interface program

============= REVISIONS ===============
Date		Version	 	Author      	Description             
----------	-------		------------  	--------------------------------------------
2019/09/27 	0000.00	 	M.Grasso		Creation of the PRG

**********************************************************************************************************)
PROGRAM _csp_case_feed_normal
VAR
END_VAR

(* CASE *)
	(* FEED *)
		(* ACCU-U-CHANGE*)
		csp_case_feed_magazine_accU();
		csp_case_feed_shuttle_accU();
		csp_case_feed_reject_accU();
		(* ARM *)
		csp_case_feed_arm();
		(* MAGAZINE *)
		csp_case_feed_magazine();
		(* REJECT *)
		csp_case_feed_reject();
		(* SHUTTLE *)
		csp_case_feed_shuttle();

		(*csp_case_feed_kinematic(); Moved to low task to manage all the axis (MCS and ACS) in the same task!

		csp_case_feed_virtualMaster();*)

END_PROGRAM

// ---- Application/CSP/Case/Feed/Arm/csp_case_feed_arm.TcPOU
(*********************************** G.D S.p.A. - Technical Department ***********************************
============= PROGRAM INFO ============
FOLDER:             TBD
MACHINES INVOLVED:  TBD 

============= DESCRIPTION =============
csp machine declaration

============= REVISIONS ===============
Date		Version	 	Author      	Description             
----------	-------		------------  	--------------------------------------------
2019/04/05 	0000.00	 	M.Grasso		Creation of the PRG

**********************************************************************************************************)
(*$R process_ref := prc; $*)
PROGRAM csp_case_feed_arm
VAR
		
	prc:											process;
	prc_path:										STRING;
END_VAR

_read_var_input();

_object_manager();

IF NOT objects_running()
THEN
	RETURN;	
END_IF

_read_process_image();

_mode_manager();

_set_runtime_properties();

(********************************* BODY *********************************)
(************************************************************************)

_handle_messages();

_write_output();

ACTION _handle_messages:
;
END_ACTION

ACTION _handle_process_test:
;
END_ACTION

ACTION _mode_manager:
IF process_mode_req_is_pending(prc)
THEN
    process_apply_mode_req_first_step(prc);
    CASE process_get_mode(prc) OF
        MODE_TO_ABSENT:
			;
        MODE_TO_INACTIVE:
			;
        MODE_TO_TEST:
			;
        MODE_TO_OPERATIONAL:
			;
    END_CASE
    process_apply_mode_req_second_step(prc);
END_IF
END_ACTION

ACTION _object_manager:
IF objects_initialization()
THEN
	sub_process_init(
		object_name					:= 'csp_case_feed_arm.prc', 
		process						:= csp_case_feed.prc, 
		CONVERSION_this				:= prc);
		
	prc_path 						:= process_get_path(prc);
END_IF

IF objects_running()
THEN
	process_cycle(prc);
END_IF
END_ACTION

ACTION _read_process_image:
;
END_ACTION

ACTION _read_var_input:
;
END_ACTION

ACTION _set_runtime_properties:
;
END_ACTION

ACTION _write_output:
;
END_ACTION

END_PROGRAM

// ---- Application/CSP/Case/Feed/Reject/csp_case_feed_reject.TcPOU
(*********************************** G.D S.p.A. - Technical Department ***********************************
============= PROGRAM INFO ============
FOLDER:             TBD
MACHINES INVOLVED:  TBD 

============= DESCRIPTION =============
csp machine declaration

============= REVISIONS ===============
Date		Version	 	Author      	Description             
----------	-------		------------  	--------------------------------------------
2019/04/05 	0000.00	 	M.Grasso		Creation of the PRG

**********************************************************************************************************)
(*$R process_ref := prc; $*)
PROGRAM csp_case_feed_reject
VAR
		
	prc:											process;
	prc_path:										STRING;
	
END_VAR

_read_var_input();

_object_manager();

IF NOT objects_running()
THEN
	RETURN;	
END_IF

_read_process_image();

_mode_manager();

_set_runtime_properties();

(********************************* BODY *********************************)
(************************************************************************)

_handle_messages();

_write_output();

ACTION _handle_messages:
;
END_ACTION

ACTION _handle_process_test:
;
END_ACTION

ACTION _mode_manager:
IF process_mode_req_is_pending(prc)
THEN
    process_apply_mode_req_first_step(prc);
    CASE process_get_mode(prc) OF
        MODE_TO_ABSENT:
			;
        MODE_TO_INACTIVE:
			;
        MODE_TO_TEST:
			;
        MODE_TO_OPERATIONAL:
			;
    END_CASE
    process_apply_mode_req_second_step(prc);
END_IF
END_ACTION

ACTION _object_manager:
IF objects_initialization()
THEN
	sub_process_init(
		object_name					:= 'csp_case_feed_reject.prc', 
		process						:= csp_case_feed.prc, 
		CONVERSION_this				:= prc);
		
	prc_path 						:= process_get_path(prc);
END_IF

IF objects_running()
THEN
	process_cycle(prc);
END_IF
END_ACTION

ACTION _read_process_image:
;
END_ACTION

ACTION _read_var_input:
;
END_ACTION

ACTION _set_runtime_properties:
;
END_ACTION

ACTION _write_output:
;
END_ACTION

END_PROGRAM

// ---- Application/CSP/Case/Feed/Shuttle/csp_case_feed_shuttle.TcPOU
(*********************************** G.D S.p.A. - Technical Department ***********************************
============= PROGRAM INFO ============
FOLDER:             TBD
MACHINES INVOLVED:  TBD 

============= DESCRIPTION =============
csp machine declaration

============= REVISIONS ===============
Date		Version	 	Author      	Description             
----------	-------		------------  	--------------------------------------------
2019/04/05 	0000.00	 	M.Grasso		Creation of the PRG

**********************************************************************************************************)
(*$R process_ref := prc; $*)
PROGRAM csp_case_feed_shuttle
VAR
	
	prc:											process;
	prc_path:										STRING;
	
END_VAR

_read_var_input();

_object_manager();

IF 	NOT objects_running()
THEN
	RETURN;	
END_IF

_read_process_image();

_mode_manager();

CASE process_get_mode(prc) OF
	MODE_ABSENT,
	MODE_INACTIVE:
		RETURN;
	MODE_TEST:
		_handle_process_test();
END_CASE

_set_runtime_properties();

(********************************* BODY *********************************)
(************************************************************************)

_handle_messages();

_write_output();

ACTION _handle_messages:
;
END_ACTION

ACTION _handle_process_test:
;
END_ACTION

ACTION _mode_manager:
IF process_mode_req_is_pending(prc)
THEN
    process_apply_mode_req_first_step(prc);
    CASE process_get_mode(prc) OF
        MODE_TO_ABSENT:
			;
        MODE_TO_INACTIVE:
			;
        MODE_TO_TEST:
			;
        MODE_TO_OPERATIONAL:
			;
    END_CASE
    process_apply_mode_req_second_step(prc);
END_IF
END_ACTION

ACTION _object_manager:
IF objects_initialization()
THEN
	sub_process_init(
		object_name					:= 'csp_case_feed_shuttle.prc', 
		process						:= csp_case_feed.prc, 
		CONVERSION_this				:= prc);
		
	prc_path 						:= process_get_path(prc);
		
END_IF

IF objects_running()
THEN
	process_cycle(prc);
END_IF
END_ACTION

ACTION _read_process_image:
;
END_ACTION

ACTION _read_var_input:
;
END_ACTION

ACTION _set_runtime_properties:
;
END_ACTION

ACTION _write_output:
;
END_ACTION

END_PROGRAM

// ---- Application/CSP/Case/Flap Control/_Tasks/_csp_case_flapControl_normal.TcPOU
(*********************************** G.D S.p.A. - Technical Department ***********************************
============= PROGRAM INFO ============
FOLDER:             TBD
MACHINES INVOLVED:  TBD 

============= DESCRIPTION =============
csp main interface program

============= REVISIONS ===============
Date		Version	 	Author      	Description             
----------	-------		------------  	--------------------------------------------
2019/09/27 	0000.00	 	M.Grasso		Creation of the PRG

**********************************************************************************************************)
PROGRAM _csp_case_flapControl_normal
VAR
END_VAR

(* CASE *)
	(* FLAP CONTROL *)
		(* BACKSTOP *)
		csp_case_flapControl_backStop();
		(* LS *)
		csp_case_flapControl_ls();
		(* OS *)
		csp_case_flapControl_os();

END_PROGRAM

// ---- Application/CSP/Case/Flap Control/Backstop/csp_case_flapControl_backStop.TcPOU
(*********************************** G.D S.p.A. - Technical Department ***********************************
============= PROGRAM INFO ============
FOLDER:             TBD
MACHINES INVOLVED:  TBD 

============= DESCRIPTION =============
csp machine declaration

============= REVISIONS ===============
Date		Version	 	Author      	Description             
----------	-------		------------  	--------------------------------------------
2019/04/05 	0000.00	 	M.Grasso		Creation of the PRG

**********************************************************************************************************)
(*$R process_ref := prc; $*)
PROGRAM csp_case_flapControl_backStop
VAR
	
	prc:											process;
	prc_path:										STRING;
	
	extend_do:										digital_output;
	extend_sact:									digital_actuator;
	present_di:										digital_input;
	
	backstop_present_lost_aem:						message;
END_VAR

_read_var_input();

_object_manager();

IF NOT objects_running()
THEN
	RETURN;	
END_IF

_read_process_image();

_mode_manager();

CASE process_get_mode(prc) OF
	MODE_ABSENT:
		digital_actuator_activate(CONVERSION_this:=extend_sact);
		digital_output_set(CONVERSION_this := extend_do);
		RETURN;
	MODE_INACTIVE:
		RETURN;
	MODE_TEST:
		_handle_process_test();
END_CASE

_set_runtime_properties();

(********************************* BODY *********************************)

IF 	csp.o_machine_is_running //(csp.mch)
	AND NOT digital_input_is_active(present_di)
THEN
	process_message_set(1,1,1, backstop_present_lost_aem);
END_IF

IF 	machine_is_stopped(csp.mch)
	OR machine_is_stop_emergency_active(csp.mch)
THEN
	process_message_reset(backstop_present_lost_aem);
END_IF


IF 	csp.o_machine_is_running
	OR
	csp.o_machine_is_ready
THEN
	digital_actuator_activate(CONVERSION_this:=extend_sact);
END_IF
(************************************************************************)

_handle_messages();

_write_output();

ACTION _handle_messages:
;
END_ACTION

ACTION _handle_process_test:
;
END_ACTION

ACTION _mode_manager:
IF process_mode_req_is_pending(prc)
THEN
    process_apply_mode_req_first_step(prc);
    CASE process_get_mode(prc) OF
        MODE_TO_ABSENT:
			;
        MODE_TO_INACTIVE:
			;
        MODE_TO_TEST:
			;
        MODE_TO_OPERATIONAL:
			;
    END_CASE
    process_apply_mode_req_second_step(prc);
END_IF
END_ACTION

ACTION _object_manager:
IF objects_initialization()
THEN
	sub_process_init(
		object_name					:= 'csp_case_flapControl_backStop.prc', 
		process						:= csp_case_flapControl.prc, 
		CONVERSION_this				:= prc);
		
	prc_path 						:= process_get_path(prc);
	
	(* OUPUTS *)
	digital_output_init(
		object_name 			:= CONCAT(prc_path, '_extend_do'),
		polarity_direct 		:= TRUE,
		process 				:= prc,
		CONVERSION_this 		:= extend_do);
	
	(* INPUTS *)
	digital_input_init(
		object_name 			:= CONCAT(prc_path, '_present_di'),
		polarity_direct 		:= TRUE,
		process 				:= prc,
		CONVERSION_this 		:= present_di);
	
	digital_actuator_init(			
		object_name					:=CONCAT(prc_path, '_extend_sact'), 
		_type           			:= DIGITAL_ACTUATOR_TYPE_IN_Ax,
		fault_reaction 				:= DIGITAL_ACTUATOR_FAULT_REACTION_IGNORE,
		active_time     			:= 2000,
		inactive_time   			:= 2000,
		dout            			:= extend_do,
		process         			:= prc,
		conversion_this 			:= extend_sact);

	digital_actuator_add_di_active(
		di_active					:=present_di,
	 	CONVERSION_this				:=extend_sact);
		
		
	process_message_init(
		object_name:= CONCAT(prc_path, '_backstop_present_lost_aem'), 
		behaviour:= MESSAGE_BEHAVIOUR_STATE, 
		reset_timeout:= 0, 
		disableable:= FALSE, 
		individual_reset:= FALSE, 
		machine_reaction:= MACHINE_REACTION_EMERGENCY_STOP, 
		typology:= MESSAGE_TYPOLOGY_EMERGENCY, 
		process:= prc, 
		CONVERSION_this:= backstop_present_lost_aem);	
	
		
END_IF

IF objects_running()
THEN
	process_cycle(prc);
	digital_actuator_cycle(extend_sact);
END_IF
END_ACTION

ACTION _read_process_image:
;
END_ACTION

ACTION _read_var_input:
;
END_ACTION

ACTION _set_runtime_properties:
;
END_ACTION

ACTION _write_output:
;
END_ACTION

END_PROGRAM

// ---- Application/CSP/Case/Flap Control/LS/csp_case_flapControl_ls.TcPOU
(*********************************** G.D S.p.A. - Technical Department ***********************************
============= PROGRAM INFO ============
FOLDER:             TBD
MACHINES INVOLVED:  TBD 

============= DESCRIPTION =============
csp machine declaration

============= REVISIONS ===============
Date		Version	 	Author      	Description             
----------	-------		------------  	--------------------------------------------
2019/04/05 	0000.00	 	M.Grasso		Creation of the PRG

**********************************************************************************************************)
(*$R process_ref := prc; $*)
PROGRAM csp_case_flapControl_ls
VAR
	
	prc:											process;
	prc_path:										STRING;
	
END_VAR

_read_var_input();

_object_manager();

IF NOT objects_running()
THEN
	RETURN;	
END_IF

_read_process_image();

_mode_manager();

_set_runtime_properties();

(********************************* BODY *********************************)
(************************************************************************)

_handle_messages();

_write_output();

ACTION _handle_messages:
;
END_ACTION

ACTION _handle_process_test:
;
END_ACTION

ACTION _mode_manager:
IF process_mode_req_is_pending(prc)
THEN
    process_apply_mode_req_first_step(prc);
    CASE process_get_mode(prc) OF
        MODE_TO_ABSENT:
			;
        MODE_TO_INACTIVE:
			;
        MODE_TO_TEST:
			;
        MODE_TO_OPERATIONAL:
			;
    END_CASE
    process_apply_mode_req_second_step(prc);
END_IF
END_ACTION

ACTION _object_manager:
IF objects_initialization()
THEN
	sub_process_init(
		object_name					:= 'csp_case_flapControl_ls.prc', 
		process						:= csp_case_flapControl.prc, 
		CONVERSION_this				:= prc);
		
	prc_path 						:= process_get_path(prc);
END_IF

IF objects_running()
THEN
	process_cycle(prc);
END_IF
END_ACTION

ACTION _read_process_image:
;
END_ACTION

ACTION _read_var_input:
;
END_ACTION

ACTION _set_runtime_properties:
;
END_ACTION

ACTION _write_output:
;
END_ACTION

END_PROGRAM

// ---- Application/CSP/Case/Flap Control/OS/csp_case_flapControl_os.TcPOU
(*********************************** G.D S.p.A. - Technical Department ***********************************
============= PROGRAM INFO ============
FOLDER:             TBD
MACHINES INVOLVED:  TBD 

============= DESCRIPTION =============
csp machine declaration

============= REVISIONS ===============
Date		Version	 	Author      	Description             
----------	-------		------------  	--------------------------------------------
2019/04/05 	0000.00	 	M.Grasso		Creation of the PRG

**********************************************************************************************************)
(*$R process_ref := prc; $*)
PROGRAM csp_case_flapControl_os
VAR
	
	prc:											process;
	prc_path:										STRING;
	
END_VAR

_read_var_input();

_object_manager();

IF NOT objects_running()
THEN
	RETURN;	
END_IF

_read_process_image();

_mode_manager();

_set_runtime_properties();

(********************************* BODY *********************************)
(************************************************************************)

_handle_messages();

_write_output();

ACTION _handle_messages:
;
END_ACTION

ACTION _handle_process_test:
;
END_ACTION

ACTION _mode_manager:
IF process_mode_req_is_pending(prc)
THEN
    process_apply_mode_req_first_step(prc);
    CASE process_get_mode(prc) OF
        MODE_TO_ABSENT:
			;
        MODE_TO_INACTIVE:
			;
        MODE_TO_TEST:
			;
        MODE_TO_OPERATIONAL:
			;
    END_CASE
    process_apply_mode_req_second_step(prc);
END_IF
END_ACTION

ACTION _object_manager:
IF objects_initialization()
THEN
	sub_process_init(
		object_name					:= 'csp_case_flapControl_os.prc', 
		process						:= csp_case_flapControl.prc, 
		CONVERSION_this				:= prc);
		
	prc_path 						:= process_get_path(prc);
END_IF

IF objects_running()
THEN
	process_cycle(prc);
END_IF
END_ACTION

ACTION _read_process_image:
;
END_ACTION

ACTION _read_var_input:
;
END_ACTION

ACTION _set_runtime_properties:
;
END_ACTION

ACTION _write_output:
;
END_ACTION

END_PROGRAM

// ---- Application/CSP/Case/Glue/_Tasks/_csp_case_glue_normal.TcPOU
(*********************************** G.D S.p.A. - Technical Department ***********************************
============= PROGRAM INFO ============
FOLDER:             TBD
MACHINES INVOLVED:  TBD 

============= DESCRIPTION =============
csp main interface program

============= REVISIONS ===============
Date		Version	 	Author      	Description             
----------	-------		------------  	--------------------------------------------
2019/09/27 	0000.00	 	M.Grasso		Creation of the PRG

**********************************************************************************************************)
PROGRAM _csp_case_glue_normal
VAR
END_VAR

(* CASE *)
	(* GLUE *)
		(* LS *)
		csp_case_glue_ls();
		(* OS *)
		csp_case_glue_os();
		(* SENSORS *)
		csp_case_glue_hotMelt_safety();

END_PROGRAM

// ---- Application/CSP/Case/Glue/LS/csp_case_glue_ls.TcPOU
(*********************************** G.D S.p.A. - Technical Department ***********************************
============= PROGRAM INFO ============
FOLDER:             TBD
MACHINES INVOLVED:  TBD 

============= DESCRIPTION =============
csp machine declaration

============= REVISIONS ===============
Date		Version	 	Author      	Description             
----------	-------		------------  	--------------------------------------------
2019/04/05 	0000.00	 	M.Grasso		Creation of the PRG

**********************************************************************************************************)
(*$R process_ref := prc; $*)
PROGRAM csp_case_glue_ls
VAR
	
	prc:											process;
	prc_path:										STRING;
	
END_VAR

_read_var_input();

_object_manager();

IF NOT objects_running()
THEN
	RETURN;	
END_IF

_read_process_image();

_mode_manager();

_set_runtime_properties();

(********************************* BODY *********************************)
(************************************************************************)

_handle_messages();

_write_output();

ACTION _handle_messages:
;
END_ACTION

ACTION _handle_process_test:
;
END_ACTION

ACTION _mode_manager:
IF process_mode_req_is_pending(prc)
THEN
    process_apply_mode_req_first_step(prc);
    CASE process_get_mode(prc) OF
        MODE_TO_ABSENT:
			;
        MODE_TO_INACTIVE:
			;
        MODE_TO_TEST:
			;
        MODE_TO_OPERATIONAL:
			;
    END_CASE
    process_apply_mode_req_second_step(prc);
END_IF
END_ACTION

ACTION _object_manager:
IF objects_initialization()
THEN
	sub_process_init(
		object_name					:= 'csp_case_glue_ls.prc', 
		process						:= csp_case_glue.prc, 
		CONVERSION_this				:= prc);
		
	prc_path 						:= process_get_path(prc);
END_IF

IF objects_running()
THEN
	process_cycle(prc);
END_IF
END_ACTION

ACTION _read_process_image:
;
END_ACTION

ACTION _read_var_input:
;
END_ACTION

ACTION _set_runtime_properties:
;
END_ACTION

ACTION _write_output:
;
END_ACTION

END_PROGRAM

// ---- Application/CSP/Case/Glue/OS/csp_case_glue_os.TcPOU
(*********************************** G.D S.p.A. - Technical Department ***********************************
============= PROGRAM INFO ============
FOLDER:             TBD
MACHINES INVOLVED:  TBD 

============= DESCRIPTION =============
csp machine declaration

============= REVISIONS ===============
Date		Version	 	Author      	Description             
----------	-------		------------  	--------------------------------------------
2019/04/05 	0000.00	 	M.Grasso		Creation of the PRG

**********************************************************************************************************)
(*$R process_ref := prc; $*)
PROGRAM csp_case_glue_os
VAR
	
	prc:											process;
	prc_path:										STRING;
	
END_VAR

_read_var_input();

_object_manager();

IF NOT objects_running()
THEN
	RETURN;	
END_IF

_read_process_image();

_mode_manager();

_set_runtime_properties();

(********************************* BODY *********************************)
(************************************************************************)

_handle_messages();

_write_output();

ACTION _handle_messages:
;
END_ACTION

ACTION _handle_process_test:
;
END_ACTION

ACTION _mode_manager:
IF process_mode_req_is_pending(prc)
THEN
    process_apply_mode_req_first_step(prc);
    CASE process_get_mode(prc) OF
        MODE_TO_ABSENT:
			;
        MODE_TO_INACTIVE:
			;
        MODE_TO_TEST:
			;
        MODE_TO_OPERATIONAL:
			;
    END_CASE
    process_apply_mode_req_second_step(prc);
END_IF
END_ACTION

ACTION _object_manager:
IF objects_initialization()
THEN
	sub_process_init(
		object_name					:= 'csp_case_glue_os.prc', 
		process						:= csp_case_glue.prc, 
		CONVERSION_this				:= prc);
		
	prc_path 						:= process_get_path(prc);
END_IF

IF objects_running()
THEN
	process_cycle(prc);
END_IF
END_ACTION

ACTION _read_process_image:
;
END_ACTION

ACTION _read_var_input:
;
END_ACTION

ACTION _set_runtime_properties:
;
END_ACTION

ACTION _write_output:
;
END_ACTION

END_PROGRAM

// ---- Application/CSP/Case/Glue/HotMelt/csp_case_glue_hotMelt_safety.TcPOU
(*********************************** G.D S.p.A. - Technical Department ***********************************
============= PROGRAM INFO ============
FOLDER:             TBD
MACHINES INVOLVED:  TBD 

============= DESCRIPTION =============
csp machine declaration

============= REVISIONS ===============
Date		Version	 	Author      	Description             
----------	-------		------------  	--------------------------------------------
2019/04/05 	0000.00	 	M.Grasso		Creation of the PRG

**********************************************************************************************************)
(*$R process_ref := prc; $*)
PROGRAM csp_case_glue_hotMelt_safety
VAR
	
	prc:											process;
	prc_path:										STRING;
	
	sig:											safety_integrated_group;
	sis:											safety_integrated_series;
END_VAR

_read_var_input();

_object_manager();

IF NOT objects_running()
THEN
	RETURN;	
END_IF

_read_process_image();

_mode_manager();

CASE process_get_mode(prc) of
	MODE_ABSENT,
	MODE_INACTIVE:
		RETURN;
	MODE_TEST:
		_handle_process_test();
END_CASE

_set_runtime_properties();

(********************************* BODY *********************************)
safety_integrated_series_close(sis);
(************************************************************************)

_handle_messages();

_write_output();

ACTION _handle_messages:
;
END_ACTION

ACTION _handle_process_test:
;
END_ACTION

ACTION _mode_manager:
IF process_mode_req_is_pending(prc)
THEN
    process_apply_mode_req_first_step(prc);
    CASE process_get_mode(prc) OF
        MODE_TO_ABSENT:
			;
        MODE_TO_INACTIVE:
			;
        MODE_TO_TEST:
			;
        MODE_TO_OPERATIONAL:
			;
    END_CASE
    process_apply_mode_req_second_step(prc);
END_IF
END_ACTION

ACTION _object_manager:
IF objects_initialization()
THEN
	sub_process_init(
		object_name						:= 'csp_case_glue_ls_guns_safety.prc', 
		process							:= csp_case_glue_ls_guns.prc, 
		CONVERSION_this					:= prc);
		
	prc_path 							:= process_get_path(prc);
	

END_IF

IF objects_running()
THEN
	process_cycle(prc);
	
END_IF
END_ACTION

ACTION _read_process_image:
;
END_ACTION

ACTION _read_var_input:
;
END_ACTION

ACTION _set_runtime_properties:
;
END_ACTION

ACTION _write_output:
;
END_ACTION

END_PROGRAM

// ---- Application/CSP/Case/Loader/_Tasks/_csp_case_loader_normal.TcPOU
(*********************************** G.D S.p.A. - Technical Department ***********************************
============= PROGRAM INFO ============
FOLDER:             TBD
MACHINES INVOLVED:  TBD 

============= DESCRIPTION =============
csp main interface program

============= REVISIONS ===============
Date		Version	 	Author      	Description             
----------	-------		------------  	--------------------------------------------
2019/09/27 	0000.00	 	M.Grasso		Creation of the PRG

**********************************************************************************************************)
PROGRAM _csp_case_loader_normal
VAR
END_VAR

(* CASE *)
	(* LOADER *)
		(* GUIDE *)
		csp_case_loader_guide();
		(* SENSORS *)
		csp_case_loader_sensors();

END_PROGRAM

// ---- Application/CSP/Case/Loader/Guide/csp_case_loader_guide.TcPOU
(*********************************** G.D S.p.A. - Technical Department ***********************************
============= PROGRAM INFO ============
FOLDER:             TBD
MACHINES INVOLVED:  TBD 

============= DESCRIPTION =============
csp machine declaration

============= REVISIONS ===============
Date		Version	 	Author      	Description             
----------	-------		------------  	--------------------------------------------
2019/04/05 	0000.00	 	M.Grasso		Creation of the PRG

**********************************************************************************************************)
(*$R process_ref := prc; $*)
PROGRAM csp_case_loader_guide
VAR
	
	prc:											process;
	prc_path:										STRING;
	
END_VAR

_read_var_input();

_object_manager();

IF NOT objects_running()
THEN
	RETURN;	
END_IF

_read_process_image();

_mode_manager();

_set_runtime_properties();

(********************************* BODY *********************************)
(************************************************************************)

_handle_messages();

_write_output();

ACTION _handle_messages:
;
END_ACTION

ACTION _handle_process_test:
;
END_ACTION

ACTION _mode_manager:
IF process_mode_req_is_pending(prc)
THEN
    process_apply_mode_req_first_step(prc);
    CASE process_get_mode(prc) OF
        MODE_TO_ABSENT:
			;
        MODE_TO_INACTIVE:
			;
        MODE_TO_TEST:
			;
        MODE_TO_OPERATIONAL:
			;
    END_CASE
    process_apply_mode_req_second_step(prc);
END_IF
END_ACTION

ACTION _object_manager:
IF objects_initialization()
THEN
	sub_process_init(
		object_name					:= 'csp_case_loader_guide.prc', 
		process						:= csp_case_loader.prc, 
		CONVERSION_this				:= prc);
		
	prc_path 						:= process_get_path(prc);
END_IF

IF objects_running()
THEN
	process_cycle(prc);
END_IF
END_ACTION

ACTION _read_process_image:
;
END_ACTION

ACTION _read_var_input:
;
END_ACTION

ACTION _set_runtime_properties:
;
END_ACTION

ACTION _write_output:
;
END_ACTION

END_PROGRAM

// ---- Application/CSP/Case/Open Flap/_Tasks/_csp_case_openFlap_normal.TcPOU
(*********************************** G.D S.p.A. - Technical Department ***********************************
============= PROGRAM INFO ============
FOLDER:             TBD
MACHINES INVOLVED:  TBD 

============= DESCRIPTION =============
csp main interface program

============= REVISIONS ===============
Date		Version	 	Author      	Description             
----------	-------		------------  	--------------------------------------------
2019/09/27 	0000.00	 	M.Grasso		Creation of the PRG

**********************************************************************************************************)
PROGRAM _csp_case_openFlap_normal
VAR
END_VAR

csp_case_openFlap_sensors();

END_PROGRAM

// ---- Application/CSP/Case/Main/_Tasks/_csp_case_main_normal.TcPOU
(*********************************** G.D S.p.A. - Technical Department ***********************************
============= PROGRAM INFO ============
FOLDER:             TBD
MACHINES INVOLVED:  TBD 

============= DESCRIPTION =============
csp main interface program

============= REVISIONS ===============
Date		Version	 	Author      	Description             
----------	-------		------------  	--------------------------------------------
2019/09/27 	0000.00	 	M.Grasso		Creation of the PRG

**********************************************************************************************************)
PROGRAM _csp_case_main_normal
VAR
END_VAR

(* MAIN *)

	(*Brand*)
	
	(*Drives*)
	csp_case_main_drives();
	(*Motorization*)

	(*Cam Manager*)
	
	(*Services*)
	csp_case_main_services();
	csp_case_main_services_airPressure();
		csp_case_main_services_vacuum();
		csp_case_main_services_pushbuttons();
		csp_case_main_services_hotMelt();
		csp_case_main_services_breakers();
		//csp_case_main_ioLink();

	(*Interface*)
	
	(*Safety*)

END_PROGRAM

// ---- Application/CSP/Case/Top Rail/_Tasks/_csp_case_topRail_normal.TcPOU
(*********************************** G.D S.p.A. - Technical Department ***********************************
============= PROGRAM INFO ============
FOLDER:             TBD
MACHINES INVOLVED:  TBD 

============= DESCRIPTION =============
csp main interface program

============= REVISIONS ===============
Date		Version	 	Author      	Description             
----------	-------		------------  	--------------------------------------------
2019/09/27 	0000.00	 	M.Grasso		Creation of the PRG

**********************************************************************************************************)
PROGRAM _csp_case_topRail_normal
VAR
END_VAR

(* CASE *)
	(* TOP RAIL *)
		(* ACC-U-CHANGE *)
		csp_case_topRail_accU();

END_PROGRAM

// ---- Application/CSP/Case/Top Rail/Acc U Change/csp_case_topRail_accU.TcPOU
(*********************************** G.D S.p.A. - Technical Department ***********************************
============= PROGRAM INFO ============
FOLDER:             TBD
MACHINES INVOLVED:  TBD 

============= DESCRIPTION =============
csp machine declaration

============= REVISIONS ===============
Date		Version	 	Author      	Description             
----------	-------		------------  	--------------------------------------------
2019/04/05 	0000.00	 	M.Grasso		Creation of the PRG

**********************************************************************************************************)
(*$R process_ref := prc; $*)
PROGRAM csp_case_topRail_accU
VAR
	
	prc:											process;
	prc_path:										STRING;
	
END_VAR

_read_var_input();

_object_manager();

IF NOT objects_running()
THEN
	RETURN;	
END_IF

_read_process_image();

_mode_manager();

_set_runtime_properties();

(********************************* BODY *********************************)
(************************************************************************)

_handle_messages();

_write_output();

ACTION _handle_messages:
;
END_ACTION

ACTION _handle_process_test:
;
END_ACTION

ACTION _mode_manager:
IF process_mode_req_is_pending(prc)
THEN
    process_apply_mode_req_first_step(prc);
    CASE process_get_mode(prc) OF
        MODE_TO_ABSENT:
			;
        MODE_TO_INACTIVE:
			;
        MODE_TO_TEST:
			;
        MODE_TO_OPERATIONAL:
			;
    END_CASE
    process_apply_mode_req_second_step(prc);
END_IF
END_ACTION

ACTION _object_manager:
IF objects_initialization()
THEN
	sub_process_init(
		object_name					:= 'csp_case_topRail_accU.prc', 
		process						:= csp_case_topRail.prc, 
		CONVERSION_this				:= prc);
		
	prc_path 						:= process_get_path(prc);
END_IF

IF objects_running()
THEN
	process_cycle(prc);
END_IF
END_ACTION

ACTION _read_process_image:
;
END_ACTION

ACTION _read_var_input:
;
END_ACTION

ACTION _set_runtime_properties:
;
END_ACTION

ACTION _write_output:
;
END_ACTION

END_PROGRAM

// ---- Application/CSP/Case/Transport/_Tasks/_csp_case_transport_normal.TcPOU
(*********************************** G.D S.p.A. - Technical Department ***********************************
============= PROGRAM INFO ============
FOLDER:             TBD
MACHINES INVOLVED:  TBD 

============= DESCRIPTION =============
csp main interface program

============= REVISIONS ===============
Date		Version	 	Author      	Description             
----------	-------		------------  	--------------------------------------------
2019/09/27 	0000.00	 	M.Grasso		Creation of the PRG

**********************************************************************************************************)
PROGRAM _csp_case_transport_normal
VAR
END_VAR

(* CSP *)
	(* TRANSPORT *)
		(* ACC-U-CHANGE *)
		csp_case_transport_accU();
		(* TENSIONER *)
		csp_case_transport_tensioner();

END_PROGRAM

// ---- Application/CSP/Case/Transport/Acc U Change/csp_case_transport_accU.TcPOU
(*********************************** G.D S.p.A. - Technical Department ***********************************
============= PROGRAM INFO ============
FOLDER:             TBD
MACHINES INVOLVED:  TBD 

============= DESCRIPTION =============
csp machine declaration

============= REVISIONS ===============
Date		Version	 	Author      	Description             
----------	-------		------------  	--------------------------------------------
2019/04/05 	0000.00	 	M.Grasso		Creation of the PRG

**********************************************************************************************************)
(*$R process_ref := prc; $*)
PROGRAM csp_case_transport_accU
VAR
	
	prc:											process;
	prc_path:										STRING;
	
END_VAR

_read_var_input();

_object_manager();

IF NOT objects_running()
THEN
	RETURN;	
END_IF

_read_process_image();

_mode_manager();
CASE process_get_mode(prc) OF
	MODE_ABSENT,
	MODE_INACTIVE:
		RETURN;
	MODE_TEST:
		_handle_process_test();
END_CASE
_set_runtime_properties();

(********************************* BODY *********************************)
(************************************************************************)

_handle_messages();

_write_output();

ACTION _handle_messages:
;
END_ACTION

ACTION _handle_process_test:
;
END_ACTION

ACTION _mode_manager:
IF process_mode_req_is_pending(prc)
THEN
    process_apply_mode_req_first_step(prc);
    CASE process_get_mode(prc) OF
        MODE_TO_ABSENT:
			;
        MODE_TO_INACTIVE:
			;
        MODE_TO_TEST:
			;
        MODE_TO_OPERATIONAL:
			;
    END_CASE
    process_apply_mode_req_second_step(prc);
END_IF
END_ACTION

ACTION _object_manager:
IF objects_initialization()
THEN
	sub_process_init(
		object_name					:= 'csp_case_transport_accU.prc', 
		process						:= csp_case_transport.prc, 
		CONVERSION_this				:= prc);
		
	prc_path 						:= process_get_path(prc);
END_IF

IF objects_running()
THEN
	process_cycle(prc);
END_IF
END_ACTION

ACTION _read_process_image:
;
END_ACTION

ACTION _read_var_input:
;
END_ACTION

ACTION _set_runtime_properties:
;
END_ACTION

ACTION _write_output:
;
END_ACTION

END_PROGRAM

// ---- Application/CSP/Case/Transport/Tensioner/csp_case_transport_tensioner.TcPOU
(*********************************** G.D S.p.A. - Technical Department ***********************************
============= PROGRAM INFO ============
FOLDER:             TBD
MACHINES INVOLVED:  TBD 

============= DESCRIPTION =============
csp machine declaration

============= REVISIONS ===============
Date		Version	 	Author      	Description             
----------	-------		------------  	--------------------------------------------
2019/04/05 	0000.00	 	M.Grasso		Creation of the PRG

**********************************************************************************************************)
(*$R process_ref := prc; $*)
PROGRAM csp_case_transport_tensioner
VAR
	
	prc:											process;
	prc_path:										STRING;
	chain_tensioner_sact:							digital_actuator;
	chain_tensioner_do:								digital_output;
	chain_tensioner_tmr:                            timer;
	
END_VAR

_read_var_input();

_object_manager();

IF NOT objects_running()
THEN
	RETURN;	
END_IF

_read_process_image();

_mode_manager();

_set_runtime_properties();

(********************************* BODY *********************************)

(* CHAIN TENSIONER SHOULD RUN ON RESET EDGE FOR 3 SECONDS THEN NOT RUN AGAIN UNTIL RESET EDGE*)
IF machine_get_reset_edge(csp.mch)
THEN
	timer_restart(
		delta_ms 		:= 3000, 
		CONVERSION_this	:= chain_tensioner_tmr);
END_IF

IF NOT timer_is_expired(chain_tensioner_tmr)
THEN	
	digital_actuator_activate(chain_tensioner_sact);
ELSE
	digital_actuator_deactivate(chain_tensioner_sact);
END_IF

(************************************************************************)

_handle_messages();

_write_output();

ACTION _handle_messages:
;
END_ACTION

ACTION _handle_process_test:
;
END_ACTION

ACTION _mode_manager:
IF process_mode_req_is_pending(prc)
THEN
    process_apply_mode_req_first_step(prc);
    CASE process_get_mode(prc) OF
        MODE_TO_ABSENT:
			;
        MODE_TO_INACTIVE:
			;
        MODE_TO_TEST:
			;
        MODE_TO_OPERATIONAL:
			;
    END_CASE
    process_apply_mode_req_second_step(prc);
END_IF
END_ACTION

ACTION _object_manager:
IF objects_initialization()
THEN
	sub_process_init(
		object_name					:= 'csp_case_transport_tensioner.prc', 
		process						:= csp_case_transport.prc, 
		CONVERSION_this				:= prc);
		
	prc_path 						:= process_get_path(prc);
	
	digital_output_init(
		object_name 				:= CONCAT(prc_path, 'chain_tensioner_do'),
		polarity_direct 			:= TRUE,
		process 					:= prc,
		CONVERSION_this 			:= chain_tensioner_do);
	timer_init(
		object_name					:= CONCAT(prc_path, 'chain_tensioner_tmr'),
		process						:=prc,
		CONVERSION_this				:=chain_tensioner_tmr );
		
	
	digital_actuator_init(			
		object_name					:=CONCAT(prc_path, '_chain_tensioner_sact'), 
		_type           			:= DIGITAL_ACTUATOR_TYPE_IN_xx,
		fault_reaction 				:= DIGITAL_ACTUATOR_FAULT_REACTION_DEACTIVATING,
		active_time     			:= 0,
		inactive_time   			:= 0,
		dout            			:= chain_tensioner_do,
		process         			:= prc,
		conversion_this 			:=chain_tensioner_sact);	
END_IF

IF objects_running()
THEN
	process_cycle(prc);
	digital_actuator_cycle(chain_tensioner_sact);
END_IF
END_ACTION

ACTION _read_process_image:
;
END_ACTION

ACTION _read_var_input:
;
END_ACTION

ACTION _set_runtime_properties:
;
END_ACTION

ACTION _write_output:
;
END_ACTION

END_PROGRAM

// ---- Application/CSP/Transfer/_Tasks/_csp_transfer_normal.TcPOU
(*********************************** G.D S.p.A. - Technical Department ***********************************
============= PROGRAM INFO ============
FOLDER:             TBD
MACHINES INVOLVED:  TBD 

============= DESCRIPTION =============
csp main interface program

============= REVISIONS ===============
Date		Version	 	Author      	Description             
----------	-------		------------  	--------------------------------------------
2019/09/27 	0000.00	 	M.Grasso		Creation of the PRG

**********************************************************************************************************)
PROGRAM _csp_transfer_normal
VAR
END_VAR

_csp_transfer_accumulator_normal();

_csp_transfer_crosspusher_normal();

_csp_transfer_main_normal();

_csp_transfer_infeed_normal();

_csp_transfer_upstacker_normal();

END_PROGRAM

// ---- Application/CSP/Transfer/Accumulator/_Tasks/_csp_transfer_accumulator_normal.TcPOU
(*********************************** G.D S.p.A. - Technical Department ***********************************
============= PROGRAM INFO ============
FOLDER:             TBD
MACHINES INVOLVED:  TBD 

============= DESCRIPTION =============
csp main interface program

============= REVISIONS ===============
Date		Version	 	Author      	Description             
----------	-------		------------  	--------------------------------------------
2019/09/27 	0000.00	 	M.Grasso		Creation of the PRG

**********************************************************************************************************)
PROGRAM _csp_transfer_accumulator_normal
VAR
END_VAR

;

END_PROGRAM

// ---- Application/CSP/Main/_Tasks/_csp_main_normal.TcPOU
(*********************************** G.D S.p.A. - Technical Department ***********************************
============= PROGRAM INFO ============
FOLDER:             TBD
MACHINES INVOLVED:  TBD 

============= DESCRIPTION =============
csp main interface program

============= REVISIONS ===============
Date		Version	 	Author      	Description             
----------	-------		------------  	--------------------------------------------
2019/09/27 	0000.00	 	M.Grasso		Creation of the PRG

**********************************************************************************************************)
PROGRAM _csp_main_normal
VAR
END_VAR

(*MAIN*)

	(* ACC-U-CHANGE *)
	csp_main_accuChange();
	
	(*Drives*)
	
	(*Motorization*)
	csp_main_motorization_speedBalance();
	(*Cam Manager*)
	
		(* PHASE MANAGER *)
		csp_main_phaseManager();
		csp_main_phaseManager_startJob();
		//csp_main_phaseManager_near_end_run();
		//csp_main_phaseManager_run_out();
		csp_main_phaseManager_end_job();
	(*Services*)
	csp_main_services();
	csp_main_services_towerLamp();
	csp_main_services_pushbuttons();
			
	(*Interface*)
	
	
	(*Safety*)
	csp_main_safety();
	csp_main_safety_interface();
	csp_main_safety_connectionShutDown();

END_PROGRAM

// ---- Application/CSP/Main/Motorization/csp_main_motorization_speedBalance.TcPOU
(*********************************** G.D S.p.A. - Technical Department ***********************************
============= PROGRAM INFO ============
FOLDER:             TBD
MACHINES INVOLVED:  TBD 

============= DESCRIPTION =============
csp main program

============= REVISIONS ===============
Date		Version	 	Author      	Description             
----------	-------		------------  	--------------------------------------------
2019/10/07 	0000.00	 	W.Gerstner		Creation of the PRG

**********************************************************************************************************)
(*$R
	process_ref := prc;
$*)
PROGRAM csp_main_motorization_speedBalance
VAR
	prc:												process;
	prc_path:											STRING;
	
	motcond:											motorization_conditioner;
	
	overspeed_ratio:									LREAL;
	overspeed_value:									LREAL;
	Overspeed_active: BOOL;
END_VAR

_read_var_input();

_object_manager();

IF NOT objects_running()
THEN
	RETURN;	
END_IF

_read_process_image();

_mode_manager();

CASE process_get_mode(prc) of
	MODE_ABSENT,
	MODE_INACTIVE:
		RETURN;
	MODE_TEST:
		_handle_process_test();
END_CASE

_set_runtime_properties();

(********************************* BODY *********************************)

overspeed_ratio := csp_main_brand.surge_case_rate_ppm / csp_main_brand.nominal_case_rate_ppm;
overspeed_value := (
						motorization_manager_get_nominal_velocity(csp_main_motorization_manager.motm)
						* 
						overspeed_ratio
					) 
					- motorization_manager_get_nominal_velocity(csp_main_motorization_manager.motm);


motorization_conditioner_set_overspeed(
			overspeed_value := overspeed_value,
			CONVERSION_this := motcond);

			
(* TO RUN MACHINE AT OVERSPEED *)
IF csp_transfer_infeed_accumulation_level.level_status = CSP_TRANSFER_INFEED_ACCUMULATION_LEVEL_STATUS_NORMAL
	OR csp_transfer_infeed_accumulation_level.level_status = CSP_TRANSFER_INFEED_ACCUMULATION_LEVEL_STATUS_JAM
	AND axis_is_moving(csp_main_motorization_virtualManager.axis)
	AND csp_main_motorization_virtualManager.axis.actual_position < 10 // USED TO VEROFY NEW SPEED IS GIVEN ONLY JUST BEFORE INDEX
THEN
	motorization_conditioner_overspeed_activate(motcond);
END_IF

(* TO TURN OFF OVERSPEED - SURGE *)
IF (
	motorization_conditioner_is_active(motcond)
	AND axis_is_moving(csp_main_motorization_virtualManager.axis)
	AND csp_main_motorization_virtualManager.axis.actual_position < 10 // USED TO VEROFY NEW SPEED IS GIVEN ONLY JUST BEFORE INDEX
	AND csp_transfer_infeed_accumulation_level.level_status < CSP_TRANSFER_INFEED_ACCUMULATION_LEVEL_STATUS_LOW
	)
	OR machine_is_stopped(csp.mch)
	OR machine_is_stop_emergency_active(csp.mch)
	OR NOT axis_is_moving(csp_main_motorization_virtualManager.axis)
THEN
	motorization_conditioner_overspeed_deactivate(motcond);
END_IF

IF motcond.status = MOTORIZATION_CONDITIONER_STATUS_OVERSPEED_ACTIVE
THEN
	Overspeed_active := TRUE;
ELSE
	Overspeed_active := FALSE;
END_IF


(************************************************************************)

_handle_messages();

_write_output();

ACTION _handle_messages:
;
END_ACTION

ACTION _handle_process_test:
;
END_ACTION

ACTION _mode_manager:
IF process_mode_req_is_pending(prc)
THEN
    process_apply_mode_req_first_step(prc);
    CASE process_get_mode(prc) OF
        MODE_TO_ABSENT:
			;
        MODE_TO_INACTIVE:
			;
        MODE_TO_TEST:
			;
        MODE_TO_OPERATIONAL:
			;
    END_CASE
    process_apply_mode_req_second_step(prc);
END_IF
END_ACTION

ACTION _object_manager:
IF objects_initialization()
THEN
	sub_process_init(
		object_name								:= 'csp_main_motorization_speedBalance.prc', 
		process									:= csp_main_motorization.prc, 
		CONVERSION_this							:= prc);
		
	prc_path 									:= process_get_path(prc);
	
	motorization_conditioner_init(
		object_name								:=	CONCAT(prc_path, '_motcond'),
		velocity_limit							:=	100.0,
		velocity_limit_active					:=	FALSE,
		idle_handshake_active					:=	FALSE,
		execute_handshake_active				:=	FALSE,
		hold_handshake_active					:=	FALSE,
		suspend_handshake_active				:=	FALSE,
		complete_handshake_active				:=	FALSE,
		abort_handshake_active					:=	FALSE,
		stop_handshake_active					:=	FALSE,
		origin									:=	MOTORIZATION_CONDITIONER_ORIGIN_INTERNAL,
		manager									:=	csp_main_motorization_manager.motm,
		process									:=	prc,
		CONVERSION_this							:=	motcond);
	
END_IF

IF objects_running()
THEN
	process_cycle(prc);
	motorization_conditioner_cycle(motcond);
END_IF
END_ACTION

ACTION _read_process_image:
;
END_ACTION

ACTION _read_var_input:
;
END_ACTION

ACTION _set_runtime_properties:
;
END_ACTION

ACTION _write_output:
;
END_ACTION

END_PROGRAM

// ---- Application/CSP/Customer Interface/_Tasks/_csp_customerInterfaces_normal.TcPOU
(*********************************** G.D S.p.A. - Technical Department ***********************************
============= PROGRAM INFO ============
FOLDER:             TBD
MACHINES INVOLVED:  TBD 

============= DESCRIPTION =============
Low task

============= REVISIONS ===============
Date		Version	 	Author      	Description             
----------	-------		------------  	--------------------------------------------
2019/03/28 	0000.00	 	CEC		 		Creation of the PRG

**********************************************************************************************************)

PROGRAM _csp_customerInterfaces_normal
VAR
END_VAR

;

END_PROGRAM

// ---- Application/CSP/Case/Main/IO Link/csp_case_main_ioLink.TcPOU
PROGRAM csp_case_main_ioLink
VAR
		prc:									process;
		prc_path:								STRING;
		
		iol_master_ep6224_IOB3030:				iol_master;
		iol_master_ep6224_IOB3020:				iol_master;
		
		
		CH1_iol_slave:							iol_slave;				(*$O ecode:= RFID2815 ;desc := Closing Guide Check OS; $*)
		CH1_iol_slave_config:					iol_slave_bis00lh_data;
		
		CH1_1_iol_slave:						iol_slave;				(*$O ecode:= RFID2800 ;desc := Loader Head Check; $*)
		CH1_1_iol_slave_config:					iol_slave_bis00lh_data;
	
		CH2_1_iol_slave:						iol_slave;				(*$O ecode:= RFID2814 ;desc := Waterfall High Load Light Curtain - Receiver; $*)
		CH2_1_iol_slave_config:					iol_slave_bis00lh_data;
		
		CH4_1_iol_slave:						iol_slave;				(*$O ecode:= PEC2803 ;desc := Waterfall High Load Light Curtain - Receiver; $*)
		CH4_1_iol_slave_config:					iol_slave_ray26p_data;
		
			(* Configuration *)
		CH1_presence_dvr:						BOOL;
		CH2_presence_dvr:						BOOL;
		CH1_1_presence_dvr:						BOOL;
		CH2_1_presence_dvr:						BOOL;
		CH4_1_presence_dvr:						BOOL;
	
		adjust_range_nvr:      					LREAL;

	(* CH1 Teach Command *)
		CH1_command_sended_dvr:					BOOL;
		CH1_setpoint_sensing_range_prow:		parameter_overwrite;

		CH1_command_teach_ok_led:				led;
		CH1_command_teach_fail_led:				led;

		CH1_teach_start_cmd_btn:				command_button;
		CH1_teach_reset_cmd_btn:  				command_button;
		
		
	(* CH1_1 Teach Command *)
		CH1_1_command_sended_dvr:				BOOL;
		CH1_1_setpoint_sensing_range_prow:		parameter_overwrite;

		CH1_1_command_teach_ok_led:				led;
		CH1_1_command_teach_fail_led:			led;

		CH1_1_teach_start_cmd_btn:				command_button;
		CH1_1_teach_reset_cmd_btn:  			command_button;

	(* CH2_1 Teach Command *)
		CH2_1_command_sended_dvr:				BOOL;
		CH2_1_setpoint_bdc1_prow:				parameter_overwrite;

		CH2_1_command_teach_ok_led:				led;
		CH2_1_command_teaching_ok_led:			led;
		CH2_1_command_teach_fail_led:			led;

		CH2_1_teach_start_cmd_btn:				command_button;
		CH2_1_teach_end_cmd_btn:  				command_button;
		CH2_1_teach_reset_cmd_btn:  			command_button;
		
	(* CH4_1 Teach Command *)
		CH4_1_command_sended_dvr:				BOOL;
		CH4_1_setpoint_bdc1_prow:				parameter_overwrite;

		CH4_1_command_teach_ok_led:				led;
		CH4_1_command_teaching_ok_led:			led;
		CH4_1_command_teach_fail_led:			led;

		CH4_1_teach_start_cmd_btn:				command_button;
		CH4_1_teach_end_cmd_btn:  				command_button;
		CH4_1_teach_reset_cmd_btn:  			command_button;
END_VAR

_read_var_input();

_object_manager();

IF NOT objects_running()
THEN
	RETURN;	
END_IF

_read_process_image();

_mode_manager();

CASE process_get_mode(prc) of
	MODE_ABSENT,
	MODE_INACTIVE:
		RETURN;
	MODE_TEST:
		_handle_process_test();
END_CASE

_set_runtime_properties();

(********************************* BODY *********************************)
(************************************************************************)

_handle_messages();

_write_output();

ACTION _handle_messages:
;
END_ACTION

ACTION _handle_process_test:
;
END_ACTION

ACTION _mode_manager:
IF process_mode_req_is_pending(prc)
THEN
    process_apply_mode_req_first_step(prc);
    CASE process_get_mode(prc) OF
        MODE_TO_ABSENT:
			;
        MODE_TO_INACTIVE:
			;
        MODE_TO_TEST:
			;
        MODE_TO_OPERATIONAL:
			;
    END_CASE
    process_apply_mode_req_second_step(prc);
END_IF
END_ACTION

ACTION _object_manager:
IF objects_initialization()
THEN
	sub_process_init(
		object_name						:= 'csp_case_main_ioLink.prc', 
		process							:= csp_case_main.prc, 
		CONVERSION_this					:= prc);
		
	prc_path 							:= process_get_path(prc);
	
		iol_master_init(
		object_name := 			'iol_master_ep6224_IOB3030',
		device_name := 			'SPLC5000Slot19',
		_type := 				IOL_MASTER_BECKHOFF_EL6224, (*AFL : EP6224 missing*)
		ethercat_master :=		csp_main.cabinet_ethercat_master,
		process := 				prc,
		CONVERSION_this := 		iol_master_ep6224_IOB3030);
		
	iol_master_init(
		object_name := 			'iol_master_ep6224_IOB3020',
		device_name := 			'SPLC5000Slot19',
		_type := 				IOL_MASTER_BECKHOFF_EL6224, (*AFL : EP6224 missing*)
		ethercat_master :=		csp_main.cabinet_ethercat_master,
		process := 				prc,
		CONVERSION_this := 		iol_master_ep6224_IOB3020);
		
		(* Channel 1 *)
	IF	CH1_presence_dvr
	THEN
		iol_slave_init(
			object_name		:= 'CH1_iol_slave',
			channel			:= IOL_MASTER_CHANNEL1,
			iol_master		:= iol_master_ep6224_IOB3030,
			process			:= prc,
			CONVERSION_this			:= CH1_iol_slave);

		iol_slave_bis00lh_configure(
			data			:= CH1_iol_slave_config,
			CONVERSION_this			:= CH1_iol_slave);

		led_init(
			object_name	:= 'CH1_command_teach_fail_led',
			process		:= prc,
			CONVERSION_this		:= CH1_command_teach_fail_led);

		led_init(
			object_name	:= 'CH1_command_teach_ok_led',
			process		:= prc,
			CONVERSION_this		:= CH1_command_teach_ok_led);

		command_button_init(
			object_name := 'CH1_teach_start_cmd_btn',
			process     := prc,
			CONVERSION_this		:= CH1_teach_start_cmd_btn);

		command_button_init(
			object_name := 'CH1_teach_reset_cmd_btn',
			process     := prc,
			CONVERSION_this		:= CH1_teach_reset_cmd_btn);

	END_IF
	
			(* Channel 1 - IOB3020*)
	IF	CH1_1_presence_dvr
	THEN
		iol_slave_init(
			object_name		:= 'CH1_1_iol_slave',
			channel			:= IOL_MASTER_CHANNEL1,
			iol_master		:= iol_master_ep6224_IOB3020,
			process			:= prc,
			CONVERSION_this			:= CH1_1_iol_slave);

		iol_slave_bis00lh_configure(
			data			:= CH1_1_iol_slave_config,
			CONVERSION_this			:= CH1_1_iol_slave);

		led_init(
			object_name	:= 'CH1_1_command_teach_fail_led',
			process		:= prc,
			CONVERSION_this		:= CH1_1_command_teach_fail_led);

		led_init(
			object_name	:= 'CH1_1_command_teach_ok_led',
			process		:= prc,
			CONVERSION_this		:= CH1_1_command_teach_ok_led);

		command_button_init(
			object_name := 'CH1_1_teach_start_cmd_btn',
			process     := prc,
			CONVERSION_this		:= CH1_1_teach_start_cmd_btn);

		command_button_init(
			object_name := 'CH1_1_teach_reset_cmd_btn',
			process     := prc,
			CONVERSION_this		:= CH1_1_teach_reset_cmd_btn);

	END_IF

		(* Channel 2  - IOB3020*)
	IF	CH2_1_presence_dvr
	THEN
		iol_slave_init(
			object_name		:= 'CH2_1_iol_slave',
			channel			:= IOL_MASTER_CHANNEL2,
			iol_master		:= iol_master_ep6224_IOB3020,
			process			:= csp_transfer.prc,
			CONVERSION_this:= CH2_1_iol_slave);

		iol_slave_bis00lh_configure(
			data			:= CH2_1_iol_slave_config,
			CONVERSION_this			:= CH2_1_iol_slave);
			
		led_init(
			object_name	:= 'CH2_1_command_teach_fail_led',
			process		:= prc,
			CONVERSION_this		:= CH2_1_command_teach_fail_led);

		led_init(
			object_name	:= 'CH2_1_command_teach_ok_led',
			process		:= prc,
			CONVERSION_this		:= CH2_1_command_teach_ok_led);

		command_button_init(
			object_name := 'CH2_1_teach_start_cmd_btn',
			process     := prc,
			CONVERSION_this		:= CH2_1_teach_start_cmd_btn);

		command_button_init(
			object_name := 'CH2_1_teach_reset_cmd_btn',
			process     := prc,
			CONVERSION_this		:= CH2_1_teach_reset_cmd_btn);

	END_IF
	
			(* Channel 4  - IOB3020*)
	IF	CH4_1_presence_dvr
	THEN
		iol_slave_init(
			object_name		:= 'CH4_1_iol_slave',
			channel			:= IOL_MASTER_CHANNEL4,
			iol_master		:= iol_master_ep6224_IOB3020,
			process			:= csp_transfer.prc,
			CONVERSION_this:= CH4_1_iol_slave);

		iol_slave_ray26p_configure(
			data			:= CH4_1_iol_slave_config,
			CONVERSION_this			:= CH4_1_iol_slave);
			
		led_init(
			object_name	:= 'CH4_1_command_teach_fail_led',
			process		:= prc,
			CONVERSION_this		:= CH4_1_command_teach_fail_led);

		led_init(
			object_name	:= 'CH4_1_command_teach_ok_led',
			process		:= prc,
			CONVERSION_this		:= CH4_1_command_teach_ok_led);

		command_button_init(
			object_name := 'CH4_1_teach_start_cmd_btn',
			process     := prc,
			CONVERSION_this		:= CH4_1_teach_start_cmd_btn);

		command_button_init(
			object_name := 'CH4_1_teach_reset_cmd_btn',
			process     := prc,
			CONVERSION_this		:= CH4_1_teach_reset_cmd_btn);

	END_IF
END_IF

IF objects_running()
THEN
	process_cycle(prc);
	iol_master_cycle(iol_master_ep6224_IOB3030);
	iol_master_cycle(iol_master_ep6224_IOB3020);
	iol_slave_cycle(CH1_iol_slave);
	iol_slave_cycle(CH1_1_iol_slave);
	iol_slave_cycle(CH2_1_iol_slave);
	iol_slave_cycle(CH4_1_iol_slave);
END_IF
END_ACTION

ACTION _read_process_image:
;
END_ACTION

ACTION _read_var_input:
;
END_ACTION

ACTION _set_runtime_properties:
;
END_ACTION

ACTION _write_output:
;
END_ACTION

END_PROGRAM

// ---- POUs/AFL extensions/IO_Link/FUN/iol_slave_bis00lh_configure.TcPOU

(*$
<p>This function configures a generic <a target="_blank" href="#iol_slave">iol_slave</a> as a <strong>Balluff BSP00UE</strong>. It allow to connect the object to the device-specific
parameters structure variable <a target="_blank" href="#iol_slave_bsp00ue_data">iol_slave_bsp00ue_data</a>.</p>
<p>This function should be called at startup only.</p>
$*)

FUNCTION iol_slave_bis00lh_configure : VOID
VAR_IN_OUT
	
	rfid_input_buffer:				iol_slave_bis00lh_pdo_input;
	rfid_input_bitheader_1:			iol_slave_bis00lh_bitheader_input;
	rfid_input_bitheader_2:			iol_slave_bis00lh_bitheader_input;
	
	rfid_output_buffer:				iol_slave_bis00lh_pdo_output;
	rfid_output_bitheader_1:			iol_slave_bis00lh_bitheader_output;
	rfid_output_bitheader_2:			iol_slave_bis00lh_bitheader_output;
	
END_VAR

VAR
	
END_VAR

